(* PLC project Regular Expressions, CODESYS CODESYS V3.5 SP18 Patch 5 *)
(* stored: creationDateTime 2024-02-02T21:46:32.2565392, version 1.1.0.0, modificationDateTime 2024-02-02T18:21:46.8982597, organization GG *)
(* Regular Expressions - this is a simple implementation.

See the documentation folder for an introduction (the folder itself). *)

{attribute 'qualified_only'}
{attribute 'strict'}
TYPE eTokenType : (INVALID := 0, LITERAL, ANYCHAR, WILDCARD);
END_TYPE

TYPE typCompiledPattern : STRUCT
  xCaseInsensitive : BOOL;
  atTokens : ARRAY[0..ParameterList.uiMaxPatternTokens] OF typPatternToken;
  uiCountTokens : UINT;
END_STRUCT;
END_TYPE

TYPE typCompiledPatternW : STRUCT
  xCaseInsensitive : BOOL;
  atTokens : ARRAY[0..ParameterList.uiMaxPatternTokens] OF typPatternTokenW;
  uiCountTokens : UINT;
END_STRUCT;
END_TYPE

TYPE typPatternToken : STRUCT
  eType : eTokenType;
  bChar : BYTE;
  bAlternativeChar : BYTE;
END_STRUCT;
END_TYPE

TYPE typPatternTokenW : STRUCT
  eType : eTokenType;
  dwChar : DWORD;
  dwAlternativeChar : DWORD;
END_STRUCT;
END_TYPE

{attribute 'parameterlist'}
{attribute 'qualified_only'}
VAR_GLOBAL CONSTANT  (* ParameterList *)
  uiMaxPatternTokens : UINT := 255;  (* The maximum amount of tokens to support parsing (compiling) - the counting starts from 0, so add 1 to the number in your mind *)
END_VAR

(* Converts an ANSI/ISO 8859-1 compiled pattern to an Unicode compiled pattern. ANSI/ISO 8859-1 compiled patterns can be converted to Unicode without any loss. *)
FUNCTION FuCompiledPatternAnsiToW : typCompiledPatternW
  VAR_INPUT
    typPattern : typCompiledPattern;
  END_VAR
  VAR
    i : UDINT;
  END_VAR

            IF typPattern.uiCountTokens = 0 THEN
    RETURN;
END_IF

FuCompiledPatternAnsiToW.xCaseInsensitive := typPattern.xCaseInsensitive;
FuCompiledPatternAnsiToW.uiCountTokens := typPattern.uiCountTokens;

FOR i := 0 TO TO_UDINT((typPattern.uiCountTokens - 1)) BY 1 DO
    FuCompiledPatternAnsiToW.atTokens[i].eType := typPattern.atTokens[i].eType;
    FuCompiledPatternAnsiToW.atTokens[i].dwChar := TO_DWORD(typPattern.atTokens[i].bChar);
    FuCompiledPatternAnsiToW.atTokens[i].dwAlternativeChar := TO_DWORD(typPattern.atTokens[i].bAlternativeChar); 
END_FOR

          
END_FUNCTION

(* Compiles the pattern into a stream of tokens for matching. The ISO 8859-1 latin alphabet can be matched case insensitive, otherwise by default the pattern is case sensitive. A few examples of valid patterns: - 'A*bEd' - 'A*?bEd' - 'A.b*e*' - '*A\.b\*e*' - 'A?\bed' The return value signifies whether compilation was successful, or the given pattern is invalid. *)
{attribute 'qualified_only'}
FUNCTION FuCompilePattern : BOOL
  VAR_INPUT
    sPattern : STRING(255);  (* The pattern string to compile *)
    xCaseInsensitive : BOOL := FALSE;  (* Whether the pattern is case insensitive (ISO 8859-1 latin1) *)
  END_VAR
  VAR_OUTPUT
    typPattern : typCompiledPattern;  (* The compiled pattern, for "FuMatchExpression" *)
  END_VAR
  VAR
    i : UINT;
    tempChar : BYTE;
    tempNextChar : BYTE;
    tempIndex : UINT;
    tempMaxStrIndex : UINT;
  END_VAR
  VAR CONSTANT
    CHAR_WILDCARD : BYTE := 42;  (* * *)
    CHAR_LAZINESS : BYTE := 63;  (* ? *)
    CHAR_DOT : BYTE := 46;  (* . *)
    CHAR_ESCAPE : BYTE := 92;  (* \ *)
  END_VAR

            FuCompilePattern := FALSE;

IF sPattern = '' THEN
    RETURN;
END_IF

tempMaxStrIndex := TO_UINT(Standard.LEN(sPattern)) - 1;

FOR i := 0 TO tempMaxStrIndex BY 1 DO
    IF sPattern[i] = 0 OR_ELSE tempIndex > ParameterList.uiMaxPatternTokens THEN
        EXIT;
    END_IF
    
    tempChar := TO_BYTE(sPattern[i]);
    
    IF i < tempMaxStrIndex THEN
        tempNextChar := TO_BYTE(sPattern[(i + 1)]);
    ELSE
        tempNextChar := 0;
    END_IF
    
    IF tempChar = CHAR_WILDCARD THEN // Wildcard (*)
        typPattern.atTokens[tempIndex].eType := eTokenType.WILDCARD;
        typPattern.atTokens[tempIndex].bChar := 0; // Use bChar as modifier to be lazy
    ELSIF
        tempChar = CHAR_LAZINESS AND_THEN
        tempIndex > 0 AND_THEN
        typPattern.atTokens[(tempIndex - 1)].eType = eTokenType.WILDCARD
    THEN // Laziness (?), but only if previously wildcard, otherwise literal
        typPattern.atTokens[(tempIndex - 1)].bChar := 1;
        CONTINUE;
    ELSIF tempChar = CHAR_DOT THEN // Single char (.)
        typPattern.atTokens[tempIndex].eType := eTokenType.ANYCHAR;
    ELSIF
        tempChar = CHAR_ESCAPE AND_THEN (
            tempNextChar = CHAR_WILDCARD OR_ELSE
            tempNextChar = CHAR_DOT
        )
    THEN // Backslash (escape token for . or *, if followed by . or *)
        typPattern.atTokens[tempIndex].eType := eTokenType.LITERAL;
        typPattern.atTokens[tempIndex].bChar := tempNextChar;
        i := i + 1;
    ELSE
        typPattern.atTokens[tempIndex].eType := eTokenType.LITERAL;
        typPattern.atTokens[tempIndex].bChar := tempChar;
        
        tempNextChar := 0;
        IF xCaseInsensitive THEN
            // Calculate for the ISO 8859-1 latin1 alphabet the uppercase or lowercase character number
            IF tempChar >= 65 AND_THEN tempChar <= 90 THEN
                // Uppercase A-Z
                tempNextChar := tempChar + 32;
            ELSIF tempChar >= 97 AND_THEN tempChar <= 122 THEN
                // Lowercase a-z
                tempNextChar := tempChar - 32;
            ELSIF tempChar >= 192 AND_THEN tempChar <= 221 AND_THEN tempChar <> 215 THEN
                // Uppercase ISO 8859-1
                tempNextChar := tempChar + 32;
            ELSIF tempChar >= 224 AND_THEN tempChar <= 253 AND_THEN tempChar <> 247 THEN
                // Lowercase ISO 8859-1
                tempNextChar := tempChar - 32; 
            END_IF
        END_IF
        
        typPattern.atTokens[tempIndex].bAlternativeChar := tempNextChar;
    END_IF
    
    tempIndex := tempIndex + 1;
    typPattern.uiCountTokens := tempIndex;
END_FOR

FuCompilePattern := (tempIndex > 0);
typPattern.xCaseInsensitive := xCaseInsensitive;

          
END_FUNCTION

(* Compiles the pattern into a stream of tokens for matching. This is the UTF-8 version of FuCompilePattern. Disabling strict conformity allows the usage of the extended ASCII alphabet (ISO 8859-1, decimal 160-255), as long as it doesn't form a valid UTF-8 byte sequence. The alphabet can be matched case insensitive, otherwise by default the pattern is case sensitive. The case mapping table is NOT completely covered, as such you MAY encounter missing case conversion for some languages. A few examples of valid patterns: - 'A*bEd' - 'A*?bEd' - 'A.b*e*' - '*A\.b\*e*' - 'A?\bed' The return value signifies whether compilation was successful, or the given pattern is invalid. *)
{attribute 'qualified_only'}
FUNCTION FuCompilePatternUTF8 : BOOL
  VAR_INPUT
    psPattern : POINTER TO STRING(1);  (* The pattern string to compile - for technical reasons this is a STRING(1), although any length is supported *)
    udiPatternLength : UDINT;  (* Pattern string length (in bytes, not codepoints) *)
    xCaseInsensitive : BOOL := FALSE;  (* Whether the pattern is case insensitive *)
    xStrictConformity : BOOL := TRUE;  (* Require strict conformity to the Unicode standard *)
  END_VAR
  VAR_OUTPUT
    typPattern : typCompiledPatternW;  (* The compiled pattern, for "FuMatchExpressionUTF8" *)
  END_VAR
  VAR
    tempPointer : POINTER TO STRING(1);
    i : UDINT;
    tempChar : DWORD;
    tempCharLength : UDINT;
    tempNextChar : DWORD;
    tempNextCharLength : UDINT;
    tempIndex : UINT;
    tempMaxStrIndex : UDINT;
  END_VAR
  VAR CONSTANT
    CHAR_WILDCARD : DWORD := 42;  (* * *)
    CHAR_LAZINESS : DWORD := 63;  (* ? *)
    CHAR_DOT : DWORD := 46;  (* . *)
    CHAR_ESCAPE : DWORD := 92;  (* \ *)
  END_VAR

            FuCompilePatternUTF8 := FALSE;

IF udiPatternLength = 0 THEN
    RETURN;
END_IF

tempPointer := psPattern;

i := 0;
tempMaxStrIndex := udiPatternLength - 1;

WHILE i <= tempMaxStrIndex DO
    IF tempIndex > ParameterList.uiMaxPatternTokens THEN
        EXIT;
    END_IF
    
    IF
        NOT FuUtf8CharToDword(
            psInput := (tempPointer + i),
            udiStringLength := (udiPatternLength - i),
            xStrictConformity := xStrictConformity,
            dwCodepoint => tempChar,
            usiByteLength => tempCharLength
        )
    THEN
        RETURN;
    END_IF
    
    IF tempChar = 0 THEN
        EXIT;
    END_IF
    
    IF
        i > tempMaxStrIndex OR_ELSE
        NOT FuUtf8CharToDword(
            psInput := (tempPointer + i + tempCharLength),
            udiStringLength := (udiPatternLength - i),
            xStrictConformity := xStrictConformity,
            dwCodepoint => tempNextChar,
            usiByteLength => tempNextCharLength
        )
    THEN
        tempNextChar := 0;
        tempNextCharLength := 0;
    END_IF
    
    IF tempChar = CHAR_WILDCARD THEN // Wildcard (*)
        typPattern.atTokens[tempIndex].eType := eTokenType.WILDCARD;
        typPattern.atTokens[tempIndex].dwChar := 0; // Use dwChar as modifier to be lazy
    ELSIF
        tempChar = CHAR_LAZINESS AND_THEN
        tempIndex > 0 AND_THEN
        typPattern.atTokens[(tempIndex - 1)].eType = eTokenType.WILDCARD
    THEN // Laziness (?), but only if previously wildcard, otherwise literal
        typPattern.atTokens[(tempIndex - 1)].dwChar := 1;
        
        i := i + tempCharLength;
        CONTINUE;
    ELSIF tempChar = CHAR_DOT THEN // Single char (.)
        typPattern.atTokens[tempIndex].eType := eTokenType.ANYCHAR;
    ELSIF
        tempChar = CHAR_ESCAPE AND_THEN (
            tempNextChar = CHAR_WILDCARD OR_ELSE
            tempNextChar = CHAR_DOT
        )
    THEN // Backslash (escape token for . or *, if followed by . or *)
        typPattern.atTokens[tempIndex].eType := eTokenType.LITERAL;
        typPattern.atTokens[tempIndex].dwChar := tempNextChar;
        i := i + tempNextCharLength;
    ELSE
        typPattern.atTokens[tempIndex].eType := eTokenType.LITERAL;
        typPattern.atTokens[tempIndex].dwChar := tempChar;
        
        IF xCaseInsensitive THEN
            // Calculate for the ISO 8859-1 latin1 alphabet the uppercase or lowercase character number (efficient way)
            IF tempChar >= 65 AND_THEN tempChar <= 90 THEN
                // Uppercase A-Z
                tempNextChar := tempChar + 32;
            ELSIF tempChar >= 97 AND_THEN tempChar <= 122 THEN
                // Lowercase a-z
                tempNextChar := tempChar - 32;
            ELSIF tempChar >= 192 AND_THEN tempChar <= 221 AND_THEN tempChar <> 215 THEN
                // Uppercase ISO 8859-1
                tempNextChar := tempChar + 32;
            ELSIF tempChar >= 224 AND_THEN tempChar <= 253 AND_THEN tempChar <> 247 THEN
                // Lowercase ISO 8859-1
                tempNextChar := tempChar - 32; 
            ELSE
                // If we're not in the ISO 8859-1 latin1 alphabet range, use the Unicode function to calculate it
                tempNextChar := FuUnicodeCodepointCaseConvert(tempChar);
            END_IF
        ELSE
            tempNextChar := 0;
        END_IF
        
        typPattern.atTokens[tempIndex].dwAlternativeChar := tempNextChar;
    END_IF
    
    tempIndex := tempIndex + 1;
    typPattern.uiCountTokens := tempIndex;
    
    i := i + tempCharLength;
END_WHILE

FuCompilePatternUTF8 := (tempIndex > 0);
typPattern.xCaseInsensitive := xCaseInsensitive;

          
END_FUNCTION

(* Compiles the pattern into a stream of tokens for matching. This is the UTF-16 (WSTRING) version of FuCompilePattern. The alphabet can be matched case insensitive, otherwise by default the pattern is case sensitive. The case mapping table is NOT completely covered, as such you MAY encounter missing case conversion for some languages. A few examples of valid patterns: - 'A*bEd' - 'A*?bEd' - 'A.b*e*' - '*A\.b\*e*' - 'A?\bed' The return value signifies whether compilation was successful, or the given pattern is invalid. *)
{attribute 'qualified_only'}
FUNCTION FuCompilePatternW : BOOL
  VAR_INPUT
    pwsPattern : POINTER TO WSTRING(1);  (* The pattern string to compile - for technical reasons this is a WSTRING(1), although any length is supported *)
    udiPatternLength : UDINT;  (* Pattern string length (in words (length in bytes/2), not codepoints) *)
    xCaseInsensitive : BOOL := FALSE;  (* Whether the pattern is case insensitive *)
  END_VAR
  VAR_OUTPUT
    typPattern : typCompiledPatternW;  (* The compiled pattern, for "FuMatchExpressionW" *)
  END_VAR
  VAR
    tempPointer : POINTER TO WSTRING(1);
    i : UDINT;
    tempChar : DWORD;
    tempCharLength : UDINT;
    tempNextChar : DWORD;
    tempNextCharLength : UDINT;
    tempIndex : UINT;
    tempMaxStrIndex : UDINT;
  END_VAR
  VAR CONSTANT
    CHAR_WILDCARD : DWORD := 42;  (* * *)
    CHAR_LAZINESS : DWORD := 63;  (* ? *)
    CHAR_DOT : DWORD := 46;  (* . *)
    CHAR_ESCAPE : DWORD := 92;  (* \ *)
  END_VAR

            FuCompilePatternW := FALSE;

IF udiPatternLength = 0 THEN
    RETURN;
END_IF

tempPointer := pwsPattern;

i := 0;
tempMaxStrIndex := udiPatternLength - 1;

WHILE i <= tempMaxStrIndex DO
    IF tempIndex > ParameterList.uiMaxPatternTokens THEN
        EXIT;
    END_IF
    
    IF NOT FuUtf16CharToDword(psInput := (tempPointer + (i * 2)), udiStringLength := (udiPatternLength - (i * 2)), dwCodepoint => tempChar, usiWordLength => tempCharLength) THEN
        RETURN;
    END_IF
    
    IF tempChar = 0 THEN
        EXIT;
    END_IF
    
    IF
        i > tempMaxStrIndex OR_ELSE
        NOT FuUtf16CharToDword(
            psInput := (tempPointer + (i * 2) + (tempCharLength * 2)),
            udiStringLength := (udiPatternLength - (i * 2) - (tempCharLength * 2)),
            dwCodepoint => tempNextChar,
            usiWordLength => tempNextCharLength
        )
    THEN
        tempNextChar := 0;
        tempNextCharLength := 0;
    END_IF
    
    IF tempChar = CHAR_WILDCARD THEN // Wildcard (*)
        typPattern.atTokens[tempIndex].eType := eTokenType.WILDCARD;
        typPattern.atTokens[tempIndex].dwChar := 0; // Use dwChar as modifier to be lazy
    ELSIF
        tempChar = CHAR_LAZINESS AND_THEN
        tempIndex > 0 AND_THEN
        typPattern.atTokens[(tempIndex - 1)].eType = eTokenType.WILDCARD
    THEN // Laziness (?), but only if previously wildcard, otherwise literal
        typPattern.atTokens[(tempIndex - 1)].dwChar := 1;
        
        i := i + tempCharLength;
        CONTINUE;
    ELSIF tempChar = CHAR_DOT THEN // Single char (.)
        typPattern.atTokens[tempIndex].eType := eTokenType.ANYCHAR;
    ELSIF
        tempChar = CHAR_ESCAPE AND_THEN (
            tempNextChar = CHAR_WILDCARD OR_ELSE
            tempNextChar = CHAR_DOT
        )
    THEN // Backslash (escape token for . or *, if followed by . or *)
        typPattern.atTokens[tempIndex].eType := eTokenType.LITERAL;
        typPattern.atTokens[tempIndex].dwChar := tempNextChar;
        i := i + tempNextCharLength;
    ELSE
        typPattern.atTokens[tempIndex].eType := eTokenType.LITERAL;
        typPattern.atTokens[tempIndex].dwChar := tempChar;
        
        IF xCaseInsensitive THEN
            // Calculate for the ISO 8859-1 latin1 alphabet the uppercase or lowercase character number (efficient way)
            IF tempChar >= 65 AND_THEN tempChar <= 90 THEN
                // Uppercase A-Z
                tempNextChar := tempChar + 32;
            ELSIF tempChar >= 97 AND_THEN tempChar <= 122 THEN
                // Lowercase a-z
                tempNextChar := tempChar - 32;
            ELSIF tempChar >= 192 AND_THEN tempChar <= 221 AND_THEN tempChar <> 215 THEN
                // Uppercase ISO 8859-1
                tempNextChar := tempChar + 32;
            ELSIF tempChar >= 224 AND_THEN tempChar <= 253 AND_THEN tempChar <> 247 THEN
                // Lowercase ISO 8859-1
                tempNextChar := tempChar - 32; 
            ELSE
                // If we're not in the ISO 8859-1 latin1 alphabet range, use the UTF-8 function to calculate it
                tempNextChar := FuUnicodeCodepointCaseConvert(tempChar);
            END_IF
        ELSE
            tempNextChar := 0;
        END_IF
        
        typPattern.atTokens[tempIndex].dwAlternativeChar := tempNextChar;
    END_IF
    
    tempIndex := tempIndex + 1;
    typPattern.uiCountTokens := tempIndex;
    
    i := i + tempCharLength;
END_WHILE

FuCompilePatternW := (tempIndex > 0);
typPattern.xCaseInsensitive := xCaseInsensitive;

          
END_FUNCTION

(* Same as FuCompilePatternW, except it doesn't take a pointer and has a fixed length. *)
{attribute 'qualified_only'}
FUNCTION FuCompilePatternW2 : BOOL
  VAR_INPUT
    wsPattern : WSTRING(255);  (* The pattern string to compile *)
    xCaseInsensitive : BOOL := FALSE;  (* Whether the pattern is case insensitive *)
  END_VAR
  VAR_OUTPUT
    typPattern : typCompiledPatternW;  (* The compiled pattern, for "FuMatchExpressionW" *)
  END_VAR

            FuCompilePatternW2 := FuCompilePatternW(ADR(wsPattern), TO_UDINT(Stu.StrLenW(ADR(wsPattern))), xCaseInsensitive, typPattern => typPattern);

          
END_FUNCTION

(* Matches the given compiled pattern against the subject. *)
{attribute 'qualified_only'}
FUNCTION FuMatchExpression : BOOL
  VAR_INPUT
    typPattern : typCompiledPattern;  (* The compiled pattern from "FuCompilePattern" *)
    psSubject : POINTER TO STRING(1);  (* A pointer to the subject string - for technical reasons this is a STRING(1), although any size is supported *)
    udiLength : UDINT;  (* The length of the subject string *)
  END_VAR
  VAR
    tempPtrStr : POINTER TO BYTE;
    tempPtrStrMatching : POINTER TO BYTE;
    tempStrIndex : UDINT;
    tempStrIndexMatching : UDINT;
    i : UINT;
    j : UINT;
    k : LINT;
    tempLaziness : BOOL;
    tempHasEndChar : BOOL;
    tempEndChar : BYTE;
    tempEndChar2 : BYTE;
    tempWildcardSearchStart : LINT;
    tempWildcardSearchEnd : LINT;
    tempWildcardSearchBy : LINT;
    tempWildcardSearchSuccess : BOOL;
  END_VAR

            FuMatchExpression := FALSE;

IF typPattern.uiCountTokens = 0 OR_ELSE udiLength = 0 THEN
    RETURN;
END_IF

tempPtrStr := psSubject;
tempStrIndex := 0;

WHILE i < typPattern.uiCountTokens DO
    IF tempStrIndex >= udiLength THEN
        // Only if all following tokens are of type WILDCARD, we can allow a match to be positive
        FOR j := i TO (typPattern.uiCountTokens - 1) BY 1 DO
            IF typPattern.atTokens[j].eType <> eTokenType.WILDCARD THEN
                FuMatchExpression := FALSE;
                RETURN;
            END_IF
        END_FOR
        
        FuMatchExpression := TRUE;
        RETURN;
    END_IF
    
    CASE typPattern.atTokens[i].eType OF
        eTokenType.INVALID: // We shouldn't ever get an invalid token inside our token array that isn't behind our count
            RETURN;
        
        eTokenType.LITERAL:
            IF
                tempPtrStr[tempStrIndex] <> typPattern.atTokens[i].bChar AND_THEN
                (
                    NOT typPattern.xCaseInsensitive OR_ELSE (
                        typPattern.atTokens[i].bAlternativeChar <> 0 AND_THEN
                        tempPtrStr[tempStrIndex] <> typPattern.atTokens[i].bAlternativeChar
                    )
                )
            THEN
                RETURN;
            END_IF
            
            tempStrIndex := tempStrIndex + 1;
        
        eTokenType.ANYCHAR:
            tempStrIndex := tempStrIndex + 1;
        
        eTokenType.WILDCARD:
            tempLaziness := (typPattern.atTokens[i].bChar = 1);
            tempHasEndChar := FALSE;
            
            FOR j := i + 1 TO (typPattern.uiCountTokens - 1) BY 1 DO
                IF typPattern.atTokens[j].eType = eTokenType.LITERAL THEN
                    tempHasEndChar := TRUE;
                    tempEndChar := typPattern.atTokens[j].bChar;
                    tempEndChar2 := typPattern.atTokens[j].bAlternativeChar;
                    EXIT;
                END_IF
            END_FOR
            
            // If we don't have any characters to match on at the end of the pattern, we match immediately
            IF NOT tempHasEndChar THEN
                FuMatchExpression := TRUE;
                RETURN;
            END_IF
            
            IF tempLaziness THEN
                // Advance token pointer once more because the next token is the laziness token we already used
                i := i + 1;
                
                // If the wildcard is lazy, search from front to back
                tempWildcardSearchStart := TO_LINT(tempStrIndex);
                tempWildcardSearchEnd := TO_LINT(udiLength);
                tempWildcardSearchBy := 1;
            ELSE
                // If the wildcard is NOT lazy, search from back to front (greedy!)
                tempWildcardSearchStart := TO_LINT(udiLength);
                tempWildcardSearchEnd := TO_LINT(tempStrIndex);
                tempWildcardSearchBy := -1;
            END_IF
            
            tempWildcardSearchSuccess := FALSE;
            FOR k := tempWildcardSearchStart TO tempWildcardSearchEnd BY tempWildcardSearchBy DO
                IF
                    tempPtrStr[k] = tempEndChar OR_ELSE
                    (typPattern.xCaseInsensitive AND_THEN tempEndChar2 <> 0 AND_THEN tempPtrStr[k] = tempEndChar2)
                THEN
                    tempWildcardSearchSuccess := TRUE;
                    tempStrIndex := TO_UDINT(k);
                    EXIT;
                END_IF
            END_FOR
            
            IF NOT tempWildcardSearchSuccess THEN
                RETURN;
            END_IF
    END_CASE
    
    i := i + 1;
END_WHILE

FuMatchExpression := (tempStrIndex >= udiLength);

          
END_FUNCTION

(* Matches the given compiled pattern against the subject. This is the UTF-8 version of FuMatchExpression. Disabling strict conformity allows the usage of the extended ASCII alphabet (ISO 8859-1, decimal 160-255), as long as it doesn't form a valid UTF-8 byte sequence. *)
{attribute 'qualified_only'}
FUNCTION FuMatchExpressionUTF8 : BOOL
  VAR_INPUT
    typPattern : typCompiledPatternW;  (* The compiled pattern from "FuCompilePatternW" *)
    psSubject : POINTER TO STRING(1);  (* A pointer to the subject string - for technical reasons this is a STRING(1), although any size is supported *)
    udiLength : UDINT;  (* The length of the subject string (in bytes, not codepoints) *)
    xStrictConformity : BOOL := TRUE;  (* Require strict conformity to the Unicode standard *)
  END_VAR
  VAR
    tempPtrStr : POINTER TO BYTE;
    tempPtrStrMatching : POINTER TO BYTE;
    tempStrIndex : UDINT;
    tempStrIndexMatching : UDINT;
    i : UINT;
    j : UINT;
    k : LINT;
    tempChar : DWORD;
    tempCharLength : USINT;
    tempNextChar : DWORD;
    tempNextCharLength : DWORD;
    tempLaziness : BOOL;
    tempHasEndChar : BOOL;
    tempEndChar : DWORD;
    tempEndChar2 : DWORD;
    tempWildcardSearchStart : LINT;
    tempWildcardSearchEnd : LINT;
    tempWildcardSearchBy : LINT;
    tempWildcardSearchOffset : UDINT;
    tempWildcardSearchSuccess : BOOL;
  END_VAR

            FuMatchExpressionUTF8 := FALSE;

IF typPattern.uiCountTokens = 0 OR_ELSE udiLength = 0 THEN
    RETURN;
END_IF

tempPtrStr := psSubject;
tempStrIndex := 0;

WHILE i < typPattern.uiCountTokens DO
    IF tempStrIndex >= udiLength THEN
        // Only if all following tokens are of type WILDCARD, we can allow a match to be positive
        FOR j := i TO (typPattern.uiCountTokens - 1) BY 1 DO
            IF typPattern.atTokens[j].eType <> eTokenType.WILDCARD THEN
                FuMatchExpressionUTF8 := FALSE;
                RETURN;
            END_IF
        END_FOR
        
        FuMatchExpressionUTF8 := TRUE;
        RETURN;
    END_IF
    
    IF
        NOT FuUtf8CharToDword(
            psInput := (tempPtrStr + tempStrIndex),
            udiStringLength := (udiLength - tempStrIndex),
            xStrictConformity := xStrictConformity,
            dwCodepoint => tempChar,
            usiByteLength => tempCharLength
        )
    THEN
        RETURN;
    END_IF
    
    CASE typPattern.atTokens[i].eType OF
        eTokenType.INVALID: // We shouldn't ever get an invalid token inside our token array that isn't behind our count
            RETURN;
        
        eTokenType.LITERAL:
            IF
                tempChar <> typPattern.atTokens[i].dwChar AND_THEN
                (
                    NOT typPattern.xCaseInsensitive OR_ELSE
                    typPattern.atTokens[i].dwAlternativeChar = 0 OR_ELSE
                    tempChar <> typPattern.atTokens[i].dwAlternativeChar
                ) 
            THEN
                RETURN;
            END_IF
            
            tempStrIndex := tempStrIndex + tempCharLength;
        
        eTokenType.ANYCHAR:
            tempStrIndex := tempStrIndex + tempCharLength;
        
        eTokenType.WILDCARD:
            tempLaziness := (typPattern.atTokens[i].dwChar = 1);
            tempHasEndChar := FALSE;
            
            FOR j := i + 1 TO (typPattern.uiCountTokens - 1) BY 1 DO
                IF typPattern.atTokens[j].eType = eTokenType.LITERAL THEN
                    tempHasEndChar := TRUE;
                    tempEndChar := typPattern.atTokens[j].dwChar;
                    tempEndChar2 := typPattern.atTokens[j].dwAlternativeChar;
                    EXIT;
                END_IF
            END_FOR
            
            // If we don't have any characters to match on at the end of the pattern, we match immediately
            IF NOT tempHasEndChar THEN
                FuMatchExpressionUTF8 := TRUE;
                RETURN;
            END_IF
            
            IF tempLaziness THEN
                // Advance token pointer once more because the next token is the laziness token we already used
                i := i + 1;
                
                // If the wildcard is lazy, search from front to back
                tempWildcardSearchStart := TO_LINT(tempStrIndex);
                tempWildcardSearchEnd := TO_LINT(udiLength);
                tempWildcardSearchBy := 1;
            ELSE
                // If the wildcard is NOT lazy, search from back to front (greedy!)
                tempWildcardSearchStart := TO_LINT(udiLength);
                tempWildcardSearchEnd := TO_LINT(tempStrIndex);
                tempWildcardSearchBy := -1;
            END_IF
            
            tempWildcardSearchSuccess := FALSE;
            tempWildcardSearchOffset := 0;
            
            FOR k := tempWildcardSearchStart TO tempWildcardSearchEnd BY tempWildcardSearchBy DO
                IF
                    FuUtf8CharToDword(
                        psInput := (tempPtrStr + LINT_TO___XWORD(k)),
                        udiStringLength := (udiLength - tempWildcardSearchOffset),
                        xStrictConformity := xStrictConformity,
                        dwCodepoint => tempNextChar,
                        usiByteLength => tempNextCharLength
                    )
                THEN
                    tempWildcardSearchOffset := tempWildcardSearchOffset + tempNextCharLength;
                    
                    IF
                        tempNextChar = tempEndChar OR_ELSE
                        (typPattern.xCaseInsensitive AND_THEN tempEndChar2 <> 0 AND_THEN tempNextChar = tempEndChar2)
                    THEN
                        tempWildcardSearchSuccess := TRUE;
                        tempStrIndex := TO_UDINT(k);
                        EXIT;
                    END_IF
                ELSE
                    tempWildcardSearchOffset := tempWildcardSearchOffset + 1;
                END_IF
            END_FOR
            
            IF NOT tempWildcardSearchSuccess THEN
                RETURN;
            END_IF
    END_CASE
    
    i := i + 1;
END_WHILE

FuMatchExpressionUTF8 := (tempStrIndex >= udiLength);

          
END_FUNCTION

(* Matches the given compiled pattern against the subject. This is the UTF-16 (WSTRING) version of FuMatchExpression. *)
{attribute 'qualified_only'}
FUNCTION FuMatchExpressionW : BOOL
  VAR_INPUT
    typPattern : typCompiledPatternW;  (* The compiled pattern from "FuCompilePatternW" *)
    pwsSubject : POINTER TO WSTRING(1);  (* A pointer to the subject string - for technical reasons this is a WSTRING(1), although any size is supported *)
    udiLength : UDINT;  (* The length of the subject string (in words (length in bytes/2), not codepoints) *)
  END_VAR
  VAR
    tempPtrStr : POINTER TO WORD;
    tempPtrStrMatching : POINTER TO WORD;
    tempStrIndex : UDINT;
    tempStrIndexMatching : UDINT;
    i : UINT;
    j : UINT;
    k : LINT;
    tempChar : DWORD;
    tempCharLength : USINT;
    tempNextChar : DWORD;
    tempNextCharLength : DWORD;
    tempLaziness : BOOL;
    tempHasEndChar : BOOL;
    tempEndChar : DWORD;
    tempEndChar2 : DWORD;
    tempWildcardSearchStart : LINT;
    tempWildcardSearchEnd : LINT;
    tempWildcardSearchBy : LINT;
    tempWildcardSearchOffset : UDINT;
    tempWildcardSearchSuccess : BOOL;
  END_VAR

            FuMatchExpressionW := FALSE;

IF typPattern.uiCountTokens = 0 OR_ELSE udiLength = 0 THEN
    RETURN;
END_IF

tempPtrStr := pwsSubject;
tempStrIndex := 0;

WHILE i < typPattern.uiCountTokens DO
    IF tempStrIndex >= udiLength THEN
        // Only if all following tokens are of type WILDCARD, we can allow a match to be positive
        FOR j := i TO (typPattern.uiCountTokens - 1) BY 1 DO
            IF typPattern.atTokens[j].eType <> eTokenType.WILDCARD THEN
                FuMatchExpressionW := FALSE;
                RETURN;
            END_IF
        END_FOR
        
        FuMatchExpressionW := TRUE;
        RETURN;
    END_IF
    
    IF NOT FuUtf16CharToDword(psInput := (tempPtrStr + (tempStrIndex * 2)), udiStringLength := (udiLength - (tempStrIndex * 2)), dwCodepoint => tempChar, usiWordLength => tempCharLength) THEN
        RETURN;
    END_IF
    
    CASE typPattern.atTokens[i].eType OF
        eTokenType.INVALID: // We shouldn't ever get an invalid token inside our token array that isn't behind our count
            RETURN;
        
        eTokenType.LITERAL:
            IF
                tempChar <> typPattern.atTokens[i].dwChar AND_THEN
                (
                    NOT typPattern.xCaseInsensitive OR_ELSE
                    typPattern.atTokens[i].dwAlternativeChar = 0 OR_ELSE
                    tempChar <> typPattern.atTokens[i].dwAlternativeChar
                ) 
            THEN
                RETURN;
            END_IF
            
            tempStrIndex := tempStrIndex + tempCharLength;
        
        eTokenType.ANYCHAR:
            tempStrIndex := tempStrIndex + tempCharLength;
        
        eTokenType.WILDCARD:
            tempLaziness := (typPattern.atTokens[i].dwChar = 1);
            tempHasEndChar := FALSE;
            
            FOR j := i + 1 TO (typPattern.uiCountTokens - 1) BY 1 DO
                IF typPattern.atTokens[j].eType = eTokenType.LITERAL THEN
                    tempHasEndChar := TRUE;
                    tempEndChar := typPattern.atTokens[j].dwChar;
                    tempEndChar2 := typPattern.atTokens[j].dwAlternativeChar;
                    EXIT;
                END_IF
            END_FOR
            
            // If we don't have any characters to match on at the end of the pattern, we match immediately
            IF NOT tempHasEndChar THEN
                FuMatchExpressionW := TRUE;
                RETURN;
            END_IF
            
            IF tempLaziness THEN
                // Advance token pointer once more because the next token is the laziness token we already used
                i := i + 1;
                
                // If the wildcard is lazy, search from front to back
                tempWildcardSearchStart := TO_LINT(tempStrIndex);
                tempWildcardSearchEnd := TO_LINT(udiLength);
                tempWildcardSearchBy := 1;
            ELSE
                // If the wildcard is NOT lazy, search from back to front (greedy!)
                tempWildcardSearchStart := TO_LINT(udiLength);
                tempWildcardSearchEnd := TO_LINT(tempStrIndex);
                tempWildcardSearchBy := -1;
            END_IF
            
            tempWildcardSearchSuccess := FALSE;
            tempWildcardSearchOffset := 0;
            
            FOR k := tempWildcardSearchStart TO tempWildcardSearchEnd BY tempWildcardSearchBy DO
                IF
                    FuUtf16CharToDword(
                        psInput := (tempPtrStr + LINT_TO___XWORD(k)),
                        udiStringLength := (udiLength - tempWildcardSearchOffset),
                        dwCodepoint => tempNextChar,
                        usiWordLength => tempNextCharLength
                    )
                THEN
                    tempWildcardSearchOffset := tempWildcardSearchOffset + tempNextCharLength;
                    
                    IF
                        tempNextChar = tempEndChar OR_ELSE
                        (typPattern.xCaseInsensitive AND_THEN tempEndChar2 <> 0 AND_THEN tempNextChar = tempEndChar2)
                    THEN
                        tempWildcardSearchSuccess := TRUE;
                        tempStrIndex := TO_UDINT(k);
                        EXIT;
                    END_IF
                ELSE
                    tempWildcardSearchOffset := tempWildcardSearchOffset + 1;
                END_IF
            END_FOR
            
            IF NOT tempWildcardSearchSuccess THEN
                RETURN;
            END_IF
    END_CASE
    
    i := i + 1;
END_WHILE

FuMatchExpressionW := (tempStrIndex >= udiLength);

          
END_FUNCTION

(* Converts the given Unicode odepoint to the lowercase or uppercase codepoint (the opposite casing). If there is no codepoint mapping, then it will return 0. *)
{attribute 'qualified_only'}
FUNCTION FuUnicodeCodepointCaseConvert : DWORD
  VAR_INPUT
    dwCodepoint : DWORD;
  END_VAR

            FuUnicodeCodepointCaseConvert := 0;

// The following code has been generated from Unicode's UnicodeData.txt file
CASE dwCodepoint OF
    65:
        FuUnicodeCodepointCaseConvert := 97;
        RETURN;
    66:
        FuUnicodeCodepointCaseConvert := 98;
        RETURN;
    67:
        FuUnicodeCodepointCaseConvert := 99;
        RETURN;
    68:
        FuUnicodeCodepointCaseConvert := 100;
        RETURN;
    69:
        FuUnicodeCodepointCaseConvert := 101;
        RETURN;
    70:
        FuUnicodeCodepointCaseConvert := 102;
        RETURN;
    71:
        FuUnicodeCodepointCaseConvert := 103;
        RETURN;
    72:
        FuUnicodeCodepointCaseConvert := 104;
        RETURN;
    73:
        FuUnicodeCodepointCaseConvert := 105;
        RETURN;
    74:
        FuUnicodeCodepointCaseConvert := 106;
        RETURN;
    75:
        FuUnicodeCodepointCaseConvert := 107;
        RETURN;
    76:
        FuUnicodeCodepointCaseConvert := 108;
        RETURN;
    77:
        FuUnicodeCodepointCaseConvert := 109;
        RETURN;
    78:
        FuUnicodeCodepointCaseConvert := 110;
        RETURN;
    79:
        FuUnicodeCodepointCaseConvert := 111;
        RETURN;
    80:
        FuUnicodeCodepointCaseConvert := 112;
        RETURN;
    81:
        FuUnicodeCodepointCaseConvert := 113;
        RETURN;
    82:
        FuUnicodeCodepointCaseConvert := 114;
        RETURN;
    83:
        FuUnicodeCodepointCaseConvert := 115;
        RETURN;
    84:
        FuUnicodeCodepointCaseConvert := 116;
        RETURN;
    85:
        FuUnicodeCodepointCaseConvert := 117;
        RETURN;
    86:
        FuUnicodeCodepointCaseConvert := 118;
        RETURN;
    87:
        FuUnicodeCodepointCaseConvert := 119;
        RETURN;
    88:
        FuUnicodeCodepointCaseConvert := 120;
        RETURN;
    89:
        FuUnicodeCodepointCaseConvert := 121;
        RETURN;
    90:
        FuUnicodeCodepointCaseConvert := 122;
        RETURN;
    97:
        FuUnicodeCodepointCaseConvert := 65;
        RETURN;
    98:
        FuUnicodeCodepointCaseConvert := 66;
        RETURN;
    99:
        FuUnicodeCodepointCaseConvert := 67;
        RETURN;
    100:
        FuUnicodeCodepointCaseConvert := 68;
        RETURN;
    101:
        FuUnicodeCodepointCaseConvert := 69;
        RETURN;
    102:
        FuUnicodeCodepointCaseConvert := 70;
        RETURN;
    103:
        FuUnicodeCodepointCaseConvert := 71;
        RETURN;
    104:
        FuUnicodeCodepointCaseConvert := 72;
        RETURN;
    105:
        FuUnicodeCodepointCaseConvert := 73;
        RETURN;
    106:
        FuUnicodeCodepointCaseConvert := 74;
        RETURN;
    107:
        FuUnicodeCodepointCaseConvert := 75;
        RETURN;
    108:
        FuUnicodeCodepointCaseConvert := 76;
        RETURN;
    109:
        FuUnicodeCodepointCaseConvert := 77;
        RETURN;
    110:
        FuUnicodeCodepointCaseConvert := 78;
        RETURN;
    111:
        FuUnicodeCodepointCaseConvert := 79;
        RETURN;
    112:
        FuUnicodeCodepointCaseConvert := 80;
        RETURN;
    113:
        FuUnicodeCodepointCaseConvert := 81;
        RETURN;
    114:
        FuUnicodeCodepointCaseConvert := 82;
        RETURN;
    115:
        FuUnicodeCodepointCaseConvert := 83;
        RETURN;
    116:
        FuUnicodeCodepointCaseConvert := 84;
        RETURN;
    117:
        FuUnicodeCodepointCaseConvert := 85;
        RETURN;
    118:
        FuUnicodeCodepointCaseConvert := 86;
        RETURN;
    119:
        FuUnicodeCodepointCaseConvert := 87;
        RETURN;
    120:
        FuUnicodeCodepointCaseConvert := 88;
        RETURN;
    121:
        FuUnicodeCodepointCaseConvert := 89;
        RETURN;
    122:
        FuUnicodeCodepointCaseConvert := 90;
        RETURN;
    181:
        FuUnicodeCodepointCaseConvert := 924;
        RETURN;
    192:
        FuUnicodeCodepointCaseConvert := 224;
        RETURN;
    193:
        FuUnicodeCodepointCaseConvert := 225;
        RETURN;
    194:
        FuUnicodeCodepointCaseConvert := 226;
        RETURN;
    195:
        FuUnicodeCodepointCaseConvert := 227;
        RETURN;
    196:
        FuUnicodeCodepointCaseConvert := 228;
        RETURN;
    197:
        FuUnicodeCodepointCaseConvert := 229;
        RETURN;
    198:
        FuUnicodeCodepointCaseConvert := 230;
        RETURN;
    199:
        FuUnicodeCodepointCaseConvert := 231;
        RETURN;
    200:
        FuUnicodeCodepointCaseConvert := 232;
        RETURN;
    201:
        FuUnicodeCodepointCaseConvert := 233;
        RETURN;
    202:
        FuUnicodeCodepointCaseConvert := 234;
        RETURN;
    203:
        FuUnicodeCodepointCaseConvert := 235;
        RETURN;
    204:
        FuUnicodeCodepointCaseConvert := 236;
        RETURN;
    205:
        FuUnicodeCodepointCaseConvert := 237;
        RETURN;
    206:
        FuUnicodeCodepointCaseConvert := 238;
        RETURN;
    207:
        FuUnicodeCodepointCaseConvert := 239;
        RETURN;
    208:
        FuUnicodeCodepointCaseConvert := 240;
        RETURN;
    209:
        FuUnicodeCodepointCaseConvert := 241;
        RETURN;
    210:
        FuUnicodeCodepointCaseConvert := 242;
        RETURN;
    211:
        FuUnicodeCodepointCaseConvert := 243;
        RETURN;
    212:
        FuUnicodeCodepointCaseConvert := 244;
        RETURN;
    213:
        FuUnicodeCodepointCaseConvert := 245;
        RETURN;
    214:
        FuUnicodeCodepointCaseConvert := 246;
        RETURN;
    216:
        FuUnicodeCodepointCaseConvert := 248;
        RETURN;
    217:
        FuUnicodeCodepointCaseConvert := 249;
        RETURN;
    218:
        FuUnicodeCodepointCaseConvert := 250;
        RETURN;
    219:
        FuUnicodeCodepointCaseConvert := 251;
        RETURN;
    220:
        FuUnicodeCodepointCaseConvert := 252;
        RETURN;
    221:
        FuUnicodeCodepointCaseConvert := 253;
        RETURN;
    222:
        FuUnicodeCodepointCaseConvert := 254;
        RETURN;
    224:
        FuUnicodeCodepointCaseConvert := 192;
        RETURN;
    225:
        FuUnicodeCodepointCaseConvert := 193;
        RETURN;
    226:
        FuUnicodeCodepointCaseConvert := 194;
        RETURN;
    227:
        FuUnicodeCodepointCaseConvert := 195;
        RETURN;
    228:
        FuUnicodeCodepointCaseConvert := 196;
        RETURN;
    229:
        FuUnicodeCodepointCaseConvert := 197;
        RETURN;
    230:
        FuUnicodeCodepointCaseConvert := 198;
        RETURN;
    231:
        FuUnicodeCodepointCaseConvert := 199;
        RETURN;
    232:
        FuUnicodeCodepointCaseConvert := 200;
        RETURN;
    233:
        FuUnicodeCodepointCaseConvert := 201;
        RETURN;
    234:
        FuUnicodeCodepointCaseConvert := 202;
        RETURN;
    235:
        FuUnicodeCodepointCaseConvert := 203;
        RETURN;
    236:
        FuUnicodeCodepointCaseConvert := 204;
        RETURN;
    237:
        FuUnicodeCodepointCaseConvert := 205;
        RETURN;
    238:
        FuUnicodeCodepointCaseConvert := 206;
        RETURN;
    239:
        FuUnicodeCodepointCaseConvert := 207;
        RETURN;
    240:
        FuUnicodeCodepointCaseConvert := 208;
        RETURN;
    241:
        FuUnicodeCodepointCaseConvert := 209;
        RETURN;
    242:
        FuUnicodeCodepointCaseConvert := 210;
        RETURN;
    243:
        FuUnicodeCodepointCaseConvert := 211;
        RETURN;
    244:
        FuUnicodeCodepointCaseConvert := 212;
        RETURN;
    245:
        FuUnicodeCodepointCaseConvert := 213;
        RETURN;
    246:
        FuUnicodeCodepointCaseConvert := 214;
        RETURN;
    248:
        FuUnicodeCodepointCaseConvert := 216;
        RETURN;
    249:
        FuUnicodeCodepointCaseConvert := 217;
        RETURN;
    250:
        FuUnicodeCodepointCaseConvert := 218;
        RETURN;
    251:
        FuUnicodeCodepointCaseConvert := 219;
        RETURN;
    252:
        FuUnicodeCodepointCaseConvert := 220;
        RETURN;
    253:
        FuUnicodeCodepointCaseConvert := 221;
        RETURN;
    254:
        FuUnicodeCodepointCaseConvert := 222;
        RETURN;
    255:
        FuUnicodeCodepointCaseConvert := 376;
        RETURN;
    256:
        FuUnicodeCodepointCaseConvert := 257;
        RETURN;
    257:
        FuUnicodeCodepointCaseConvert := 256;
        RETURN;
    258:
        FuUnicodeCodepointCaseConvert := 259;
        RETURN;
    259:
        FuUnicodeCodepointCaseConvert := 258;
        RETURN;
    260:
        FuUnicodeCodepointCaseConvert := 261;
        RETURN;
    261:
        FuUnicodeCodepointCaseConvert := 260;
        RETURN;
    262:
        FuUnicodeCodepointCaseConvert := 263;
        RETURN;
    263:
        FuUnicodeCodepointCaseConvert := 262;
        RETURN;
    264:
        FuUnicodeCodepointCaseConvert := 265;
        RETURN;
    265:
        FuUnicodeCodepointCaseConvert := 264;
        RETURN;
    266:
        FuUnicodeCodepointCaseConvert := 267;
        RETURN;
    267:
        FuUnicodeCodepointCaseConvert := 266;
        RETURN;
    268:
        FuUnicodeCodepointCaseConvert := 269;
        RETURN;
    269:
        FuUnicodeCodepointCaseConvert := 268;
        RETURN;
    270:
        FuUnicodeCodepointCaseConvert := 271;
        RETURN;
    271:
        FuUnicodeCodepointCaseConvert := 270;
        RETURN;
    272:
        FuUnicodeCodepointCaseConvert := 273;
        RETURN;
    273:
        FuUnicodeCodepointCaseConvert := 272;
        RETURN;
    274:
        FuUnicodeCodepointCaseConvert := 275;
        RETURN;
    275:
        FuUnicodeCodepointCaseConvert := 274;
        RETURN;
    276:
        FuUnicodeCodepointCaseConvert := 277;
        RETURN;
    277:
        FuUnicodeCodepointCaseConvert := 276;
        RETURN;
    278:
        FuUnicodeCodepointCaseConvert := 279;
        RETURN;
    279:
        FuUnicodeCodepointCaseConvert := 278;
        RETURN;
    280:
        FuUnicodeCodepointCaseConvert := 281;
        RETURN;
    281:
        FuUnicodeCodepointCaseConvert := 280;
        RETURN;
    282:
        FuUnicodeCodepointCaseConvert := 283;
        RETURN;
    283:
        FuUnicodeCodepointCaseConvert := 282;
        RETURN;
    284:
        FuUnicodeCodepointCaseConvert := 285;
        RETURN;
    285:
        FuUnicodeCodepointCaseConvert := 284;
        RETURN;
    286:
        FuUnicodeCodepointCaseConvert := 287;
        RETURN;
    287:
        FuUnicodeCodepointCaseConvert := 286;
        RETURN;
    288:
        FuUnicodeCodepointCaseConvert := 289;
        RETURN;
    289:
        FuUnicodeCodepointCaseConvert := 288;
        RETURN;
    290:
        FuUnicodeCodepointCaseConvert := 291;
        RETURN;
    291:
        FuUnicodeCodepointCaseConvert := 290;
        RETURN;
    292:
        FuUnicodeCodepointCaseConvert := 293;
        RETURN;
    293:
        FuUnicodeCodepointCaseConvert := 292;
        RETURN;
    294:
        FuUnicodeCodepointCaseConvert := 295;
        RETURN;
    295:
        FuUnicodeCodepointCaseConvert := 294;
        RETURN;
    296:
        FuUnicodeCodepointCaseConvert := 297;
        RETURN;
    297:
        FuUnicodeCodepointCaseConvert := 296;
        RETURN;
    298:
        FuUnicodeCodepointCaseConvert := 299;
        RETURN;
    299:
        FuUnicodeCodepointCaseConvert := 298;
        RETURN;
    300:
        FuUnicodeCodepointCaseConvert := 301;
        RETURN;
    301:
        FuUnicodeCodepointCaseConvert := 300;
        RETURN;
    302:
        FuUnicodeCodepointCaseConvert := 303;
        RETURN;
    303:
        FuUnicodeCodepointCaseConvert := 302;
        RETURN;
    304:
        FuUnicodeCodepointCaseConvert := 105;
        RETURN;
    305:
        FuUnicodeCodepointCaseConvert := 73;
        RETURN;
    306:
        FuUnicodeCodepointCaseConvert := 307;
        RETURN;
    307:
        FuUnicodeCodepointCaseConvert := 306;
        RETURN;
    308:
        FuUnicodeCodepointCaseConvert := 309;
        RETURN;
    309:
        FuUnicodeCodepointCaseConvert := 308;
        RETURN;
    310:
        FuUnicodeCodepointCaseConvert := 311;
        RETURN;
    311:
        FuUnicodeCodepointCaseConvert := 310;
        RETURN;
    313:
        FuUnicodeCodepointCaseConvert := 314;
        RETURN;
    314:
        FuUnicodeCodepointCaseConvert := 313;
        RETURN;
    315:
        FuUnicodeCodepointCaseConvert := 316;
        RETURN;
    316:
        FuUnicodeCodepointCaseConvert := 315;
        RETURN;
    317:
        FuUnicodeCodepointCaseConvert := 318;
        RETURN;
    318:
        FuUnicodeCodepointCaseConvert := 317;
        RETURN;
    319:
        FuUnicodeCodepointCaseConvert := 320;
        RETURN;
    320:
        FuUnicodeCodepointCaseConvert := 319;
        RETURN;
    321:
        FuUnicodeCodepointCaseConvert := 322;
        RETURN;
    322:
        FuUnicodeCodepointCaseConvert := 321;
        RETURN;
    323:
        FuUnicodeCodepointCaseConvert := 324;
        RETURN;
    324:
        FuUnicodeCodepointCaseConvert := 323;
        RETURN;
    325:
        FuUnicodeCodepointCaseConvert := 326;
        RETURN;
    326:
        FuUnicodeCodepointCaseConvert := 325;
        RETURN;
    327:
        FuUnicodeCodepointCaseConvert := 328;
        RETURN;
    328:
        FuUnicodeCodepointCaseConvert := 327;
        RETURN;
    330:
        FuUnicodeCodepointCaseConvert := 331;
        RETURN;
    331:
        FuUnicodeCodepointCaseConvert := 330;
        RETURN;
    332:
        FuUnicodeCodepointCaseConvert := 333;
        RETURN;
    333:
        FuUnicodeCodepointCaseConvert := 332;
        RETURN;
    334:
        FuUnicodeCodepointCaseConvert := 335;
        RETURN;
    335:
        FuUnicodeCodepointCaseConvert := 334;
        RETURN;
    336:
        FuUnicodeCodepointCaseConvert := 337;
        RETURN;
    337:
        FuUnicodeCodepointCaseConvert := 336;
        RETURN;
    338:
        FuUnicodeCodepointCaseConvert := 339;
        RETURN;
    339:
        FuUnicodeCodepointCaseConvert := 338;
        RETURN;
    340:
        FuUnicodeCodepointCaseConvert := 341;
        RETURN;
    341:
        FuUnicodeCodepointCaseConvert := 340;
        RETURN;
    342:
        FuUnicodeCodepointCaseConvert := 343;
        RETURN;
    343:
        FuUnicodeCodepointCaseConvert := 342;
        RETURN;
    344:
        FuUnicodeCodepointCaseConvert := 345;
        RETURN;
    345:
        FuUnicodeCodepointCaseConvert := 344;
        RETURN;
    346:
        FuUnicodeCodepointCaseConvert := 347;
        RETURN;
    347:
        FuUnicodeCodepointCaseConvert := 346;
        RETURN;
    348:
        FuUnicodeCodepointCaseConvert := 349;
        RETURN;
    349:
        FuUnicodeCodepointCaseConvert := 348;
        RETURN;
    350:
        FuUnicodeCodepointCaseConvert := 351;
        RETURN;
    351:
        FuUnicodeCodepointCaseConvert := 350;
        RETURN;
    352:
        FuUnicodeCodepointCaseConvert := 353;
        RETURN;
    353:
        FuUnicodeCodepointCaseConvert := 352;
        RETURN;
    354:
        FuUnicodeCodepointCaseConvert := 355;
        RETURN;
    355:
        FuUnicodeCodepointCaseConvert := 354;
        RETURN;
    356:
        FuUnicodeCodepointCaseConvert := 357;
        RETURN;
    357:
        FuUnicodeCodepointCaseConvert := 356;
        RETURN;
    358:
        FuUnicodeCodepointCaseConvert := 359;
        RETURN;
    359:
        FuUnicodeCodepointCaseConvert := 358;
        RETURN;
    360:
        FuUnicodeCodepointCaseConvert := 361;
        RETURN;
    361:
        FuUnicodeCodepointCaseConvert := 360;
        RETURN;
    362:
        FuUnicodeCodepointCaseConvert := 363;
        RETURN;
    363:
        FuUnicodeCodepointCaseConvert := 362;
        RETURN;
    364:
        FuUnicodeCodepointCaseConvert := 365;
        RETURN;
    365:
        FuUnicodeCodepointCaseConvert := 364;
        RETURN;
    366:
        FuUnicodeCodepointCaseConvert := 367;
        RETURN;
    367:
        FuUnicodeCodepointCaseConvert := 366;
        RETURN;
    368:
        FuUnicodeCodepointCaseConvert := 369;
        RETURN;
    369:
        FuUnicodeCodepointCaseConvert := 368;
        RETURN;
    370:
        FuUnicodeCodepointCaseConvert := 371;
        RETURN;
    371:
        FuUnicodeCodepointCaseConvert := 370;
        RETURN;
    372:
        FuUnicodeCodepointCaseConvert := 373;
        RETURN;
    373:
        FuUnicodeCodepointCaseConvert := 372;
        RETURN;
    374:
        FuUnicodeCodepointCaseConvert := 375;
        RETURN;
    375:
        FuUnicodeCodepointCaseConvert := 374;
        RETURN;
    376:
        FuUnicodeCodepointCaseConvert := 255;
        RETURN;
    377:
        FuUnicodeCodepointCaseConvert := 378;
        RETURN;
    378:
        FuUnicodeCodepointCaseConvert := 377;
        RETURN;
    379:
        FuUnicodeCodepointCaseConvert := 380;
        RETURN;
    380:
        FuUnicodeCodepointCaseConvert := 379;
        RETURN;
    381:
        FuUnicodeCodepointCaseConvert := 382;
        RETURN;
    382:
        FuUnicodeCodepointCaseConvert := 381;
        RETURN;
    383:
        FuUnicodeCodepointCaseConvert := 83;
        RETURN;
    384:
        FuUnicodeCodepointCaseConvert := 579;
        RETURN;
    385:
        FuUnicodeCodepointCaseConvert := 595;
        RETURN;
    386:
        FuUnicodeCodepointCaseConvert := 387;
        RETURN;
    387:
        FuUnicodeCodepointCaseConvert := 386;
        RETURN;
    388:
        FuUnicodeCodepointCaseConvert := 389;
        RETURN;
    389:
        FuUnicodeCodepointCaseConvert := 388;
        RETURN;
    390:
        FuUnicodeCodepointCaseConvert := 596;
        RETURN;
    391:
        FuUnicodeCodepointCaseConvert := 392;
        RETURN;
    392:
        FuUnicodeCodepointCaseConvert := 391;
        RETURN;
    393:
        FuUnicodeCodepointCaseConvert := 598;
        RETURN;
    394:
        FuUnicodeCodepointCaseConvert := 599;
        RETURN;
    395:
        FuUnicodeCodepointCaseConvert := 396;
        RETURN;
    396:
        FuUnicodeCodepointCaseConvert := 395;
        RETURN;
    398:
        FuUnicodeCodepointCaseConvert := 477;
        RETURN;
    399:
        FuUnicodeCodepointCaseConvert := 601;
        RETURN;
    400:
        FuUnicodeCodepointCaseConvert := 603;
        RETURN;
    401:
        FuUnicodeCodepointCaseConvert := 402;
        RETURN;
    402:
        FuUnicodeCodepointCaseConvert := 401;
        RETURN;
    403:
        FuUnicodeCodepointCaseConvert := 608;
        RETURN;
    404:
        FuUnicodeCodepointCaseConvert := 611;
        RETURN;
    405:
        FuUnicodeCodepointCaseConvert := 502;
        RETURN;
    406:
        FuUnicodeCodepointCaseConvert := 617;
        RETURN;
    407:
        FuUnicodeCodepointCaseConvert := 616;
        RETURN;
    408:
        FuUnicodeCodepointCaseConvert := 409;
        RETURN;
    409:
        FuUnicodeCodepointCaseConvert := 408;
        RETURN;
    410:
        FuUnicodeCodepointCaseConvert := 573;
        RETURN;
    412:
        FuUnicodeCodepointCaseConvert := 623;
        RETURN;
    413:
        FuUnicodeCodepointCaseConvert := 626;
        RETURN;
    414:
        FuUnicodeCodepointCaseConvert := 544;
        RETURN;
    415:
        FuUnicodeCodepointCaseConvert := 629;
        RETURN;
    416:
        FuUnicodeCodepointCaseConvert := 417;
        RETURN;
    417:
        FuUnicodeCodepointCaseConvert := 416;
        RETURN;
    418:
        FuUnicodeCodepointCaseConvert := 419;
        RETURN;
    419:
        FuUnicodeCodepointCaseConvert := 418;
        RETURN;
    420:
        FuUnicodeCodepointCaseConvert := 421;
        RETURN;
    421:
        FuUnicodeCodepointCaseConvert := 420;
        RETURN;
    422:
        FuUnicodeCodepointCaseConvert := 640;
        RETURN;
    423:
        FuUnicodeCodepointCaseConvert := 424;
        RETURN;
    424:
        FuUnicodeCodepointCaseConvert := 423;
        RETURN;
    425:
        FuUnicodeCodepointCaseConvert := 643;
        RETURN;
    428:
        FuUnicodeCodepointCaseConvert := 429;
        RETURN;
    429:
        FuUnicodeCodepointCaseConvert := 428;
        RETURN;
    430:
        FuUnicodeCodepointCaseConvert := 648;
        RETURN;
    431:
        FuUnicodeCodepointCaseConvert := 432;
        RETURN;
    432:
        FuUnicodeCodepointCaseConvert := 431;
        RETURN;
    433:
        FuUnicodeCodepointCaseConvert := 650;
        RETURN;
    434:
        FuUnicodeCodepointCaseConvert := 651;
        RETURN;
    435:
        FuUnicodeCodepointCaseConvert := 436;
        RETURN;
    436:
        FuUnicodeCodepointCaseConvert := 435;
        RETURN;
    437:
        FuUnicodeCodepointCaseConvert := 438;
        RETURN;
    438:
        FuUnicodeCodepointCaseConvert := 437;
        RETURN;
    439:
        FuUnicodeCodepointCaseConvert := 658;
        RETURN;
    440:
        FuUnicodeCodepointCaseConvert := 441;
        RETURN;
    441:
        FuUnicodeCodepointCaseConvert := 440;
        RETURN;
    444:
        FuUnicodeCodepointCaseConvert := 445;
        RETURN;
    445:
        FuUnicodeCodepointCaseConvert := 444;
        RETURN;
    447:
        FuUnicodeCodepointCaseConvert := 503;
        RETURN;
    452:
        FuUnicodeCodepointCaseConvert := 453;
        RETURN;
    453:
        FuUnicodeCodepointCaseConvert := 453;
        RETURN;
    454:
        FuUnicodeCodepointCaseConvert := 453;
        RETURN;
    455:
        FuUnicodeCodepointCaseConvert := 456;
        RETURN;
    456:
        FuUnicodeCodepointCaseConvert := 456;
        RETURN;
    457:
        FuUnicodeCodepointCaseConvert := 456;
        RETURN;
    458:
        FuUnicodeCodepointCaseConvert := 459;
        RETURN;
    459:
        FuUnicodeCodepointCaseConvert := 459;
        RETURN;
    460:
        FuUnicodeCodepointCaseConvert := 459;
        RETURN;
    461:
        FuUnicodeCodepointCaseConvert := 462;
        RETURN;
    462:
        FuUnicodeCodepointCaseConvert := 461;
        RETURN;
    463:
        FuUnicodeCodepointCaseConvert := 464;
        RETURN;
    464:
        FuUnicodeCodepointCaseConvert := 463;
        RETURN;
    465:
        FuUnicodeCodepointCaseConvert := 466;
        RETURN;
    466:
        FuUnicodeCodepointCaseConvert := 465;
        RETURN;
    467:
        FuUnicodeCodepointCaseConvert := 468;
        RETURN;
    468:
        FuUnicodeCodepointCaseConvert := 467;
        RETURN;
    469:
        FuUnicodeCodepointCaseConvert := 470;
        RETURN;
    470:
        FuUnicodeCodepointCaseConvert := 469;
        RETURN;
    471:
        FuUnicodeCodepointCaseConvert := 472;
        RETURN;
    472:
        FuUnicodeCodepointCaseConvert := 471;
        RETURN;
    473:
        FuUnicodeCodepointCaseConvert := 474;
        RETURN;
    474:
        FuUnicodeCodepointCaseConvert := 473;
        RETURN;
    475:
        FuUnicodeCodepointCaseConvert := 476;
        RETURN;
    476:
        FuUnicodeCodepointCaseConvert := 475;
        RETURN;
    477:
        FuUnicodeCodepointCaseConvert := 398;
        RETURN;
    478:
        FuUnicodeCodepointCaseConvert := 479;
        RETURN;
    479:
        FuUnicodeCodepointCaseConvert := 478;
        RETURN;
    480:
        FuUnicodeCodepointCaseConvert := 481;
        RETURN;
    481:
        FuUnicodeCodepointCaseConvert := 480;
        RETURN;
    482:
        FuUnicodeCodepointCaseConvert := 483;
        RETURN;
    483:
        FuUnicodeCodepointCaseConvert := 482;
        RETURN;
    484:
        FuUnicodeCodepointCaseConvert := 485;
        RETURN;
    485:
        FuUnicodeCodepointCaseConvert := 484;
        RETURN;
    486:
        FuUnicodeCodepointCaseConvert := 487;
        RETURN;
    487:
        FuUnicodeCodepointCaseConvert := 486;
        RETURN;
    488:
        FuUnicodeCodepointCaseConvert := 489;
        RETURN;
    489:
        FuUnicodeCodepointCaseConvert := 488;
        RETURN;
    490:
        FuUnicodeCodepointCaseConvert := 491;
        RETURN;
    491:
        FuUnicodeCodepointCaseConvert := 490;
        RETURN;
    492:
        FuUnicodeCodepointCaseConvert := 493;
        RETURN;
    493:
        FuUnicodeCodepointCaseConvert := 492;
        RETURN;
    494:
        FuUnicodeCodepointCaseConvert := 495;
        RETURN;
    495:
        FuUnicodeCodepointCaseConvert := 494;
        RETURN;
    497:
        FuUnicodeCodepointCaseConvert := 498;
        RETURN;
    498:
        FuUnicodeCodepointCaseConvert := 498;
        RETURN;
    499:
        FuUnicodeCodepointCaseConvert := 498;
        RETURN;
    500:
        FuUnicodeCodepointCaseConvert := 501;
        RETURN;
    501:
        FuUnicodeCodepointCaseConvert := 500;
        RETURN;
    502:
        FuUnicodeCodepointCaseConvert := 405;
        RETURN;
    503:
        FuUnicodeCodepointCaseConvert := 447;
        RETURN;
    504:
        FuUnicodeCodepointCaseConvert := 505;
        RETURN;
    505:
        FuUnicodeCodepointCaseConvert := 504;
        RETURN;
    506:
        FuUnicodeCodepointCaseConvert := 507;
        RETURN;
    507:
        FuUnicodeCodepointCaseConvert := 506;
        RETURN;
    508:
        FuUnicodeCodepointCaseConvert := 509;
        RETURN;
    509:
        FuUnicodeCodepointCaseConvert := 508;
        RETURN;
    510:
        FuUnicodeCodepointCaseConvert := 511;
        RETURN;
    511:
        FuUnicodeCodepointCaseConvert := 510;
        RETURN;
    512:
        FuUnicodeCodepointCaseConvert := 513;
        RETURN;
    513:
        FuUnicodeCodepointCaseConvert := 512;
        RETURN;
    514:
        FuUnicodeCodepointCaseConvert := 515;
        RETURN;
    515:
        FuUnicodeCodepointCaseConvert := 514;
        RETURN;
    516:
        FuUnicodeCodepointCaseConvert := 517;
        RETURN;
    517:
        FuUnicodeCodepointCaseConvert := 516;
        RETURN;
    518:
        FuUnicodeCodepointCaseConvert := 519;
        RETURN;
    519:
        FuUnicodeCodepointCaseConvert := 518;
        RETURN;
    520:
        FuUnicodeCodepointCaseConvert := 521;
        RETURN;
    521:
        FuUnicodeCodepointCaseConvert := 520;
        RETURN;
    522:
        FuUnicodeCodepointCaseConvert := 523;
        RETURN;
    523:
        FuUnicodeCodepointCaseConvert := 522;
        RETURN;
    524:
        FuUnicodeCodepointCaseConvert := 525;
        RETURN;
    525:
        FuUnicodeCodepointCaseConvert := 524;
        RETURN;
    526:
        FuUnicodeCodepointCaseConvert := 527;
        RETURN;
    527:
        FuUnicodeCodepointCaseConvert := 526;
        RETURN;
    528:
        FuUnicodeCodepointCaseConvert := 529;
        RETURN;
    529:
        FuUnicodeCodepointCaseConvert := 528;
        RETURN;
    530:
        FuUnicodeCodepointCaseConvert := 531;
        RETURN;
    531:
        FuUnicodeCodepointCaseConvert := 530;
        RETURN;
    532:
        FuUnicodeCodepointCaseConvert := 533;
        RETURN;
    533:
        FuUnicodeCodepointCaseConvert := 532;
        RETURN;
    534:
        FuUnicodeCodepointCaseConvert := 535;
        RETURN;
    535:
        FuUnicodeCodepointCaseConvert := 534;
        RETURN;
    536:
        FuUnicodeCodepointCaseConvert := 537;
        RETURN;
    537:
        FuUnicodeCodepointCaseConvert := 536;
        RETURN;
    538:
        FuUnicodeCodepointCaseConvert := 539;
        RETURN;
    539:
        FuUnicodeCodepointCaseConvert := 538;
        RETURN;
    540:
        FuUnicodeCodepointCaseConvert := 541;
        RETURN;
    541:
        FuUnicodeCodepointCaseConvert := 540;
        RETURN;
    542:
        FuUnicodeCodepointCaseConvert := 543;
        RETURN;
    543:
        FuUnicodeCodepointCaseConvert := 542;
        RETURN;
    544:
        FuUnicodeCodepointCaseConvert := 414;
        RETURN;
    546:
        FuUnicodeCodepointCaseConvert := 547;
        RETURN;
    547:
        FuUnicodeCodepointCaseConvert := 546;
        RETURN;
    548:
        FuUnicodeCodepointCaseConvert := 549;
        RETURN;
    549:
        FuUnicodeCodepointCaseConvert := 548;
        RETURN;
    550:
        FuUnicodeCodepointCaseConvert := 551;
        RETURN;
    551:
        FuUnicodeCodepointCaseConvert := 550;
        RETURN;
    552:
        FuUnicodeCodepointCaseConvert := 553;
        RETURN;
    553:
        FuUnicodeCodepointCaseConvert := 552;
        RETURN;
    554:
        FuUnicodeCodepointCaseConvert := 555;
        RETURN;
    555:
        FuUnicodeCodepointCaseConvert := 554;
        RETURN;
    556:
        FuUnicodeCodepointCaseConvert := 557;
        RETURN;
    557:
        FuUnicodeCodepointCaseConvert := 556;
        RETURN;
    558:
        FuUnicodeCodepointCaseConvert := 559;
        RETURN;
    559:
        FuUnicodeCodepointCaseConvert := 558;
        RETURN;
    560:
        FuUnicodeCodepointCaseConvert := 561;
        RETURN;
    561:
        FuUnicodeCodepointCaseConvert := 560;
        RETURN;
    562:
        FuUnicodeCodepointCaseConvert := 563;
        RETURN;
    563:
        FuUnicodeCodepointCaseConvert := 562;
        RETURN;
    570:
        FuUnicodeCodepointCaseConvert := 11365;
        RETURN;
    571:
        FuUnicodeCodepointCaseConvert := 572;
        RETURN;
    572:
        FuUnicodeCodepointCaseConvert := 571;
        RETURN;
    573:
        FuUnicodeCodepointCaseConvert := 410;
        RETURN;
    574:
        FuUnicodeCodepointCaseConvert := 11366;
        RETURN;
    575:
        FuUnicodeCodepointCaseConvert := 11390;
        RETURN;
    576:
        FuUnicodeCodepointCaseConvert := 11391;
        RETURN;
    577:
        FuUnicodeCodepointCaseConvert := 578;
        RETURN;
    578:
        FuUnicodeCodepointCaseConvert := 577;
        RETURN;
    579:
        FuUnicodeCodepointCaseConvert := 384;
        RETURN;
    580:
        FuUnicodeCodepointCaseConvert := 649;
        RETURN;
    581:
        FuUnicodeCodepointCaseConvert := 652;
        RETURN;
    582:
        FuUnicodeCodepointCaseConvert := 583;
        RETURN;
    583:
        FuUnicodeCodepointCaseConvert := 582;
        RETURN;
    584:
        FuUnicodeCodepointCaseConvert := 585;
        RETURN;
    585:
        FuUnicodeCodepointCaseConvert := 584;
        RETURN;
    586:
        FuUnicodeCodepointCaseConvert := 587;
        RETURN;
    587:
        FuUnicodeCodepointCaseConvert := 586;
        RETURN;
    588:
        FuUnicodeCodepointCaseConvert := 589;
        RETURN;
    589:
        FuUnicodeCodepointCaseConvert := 588;
        RETURN;
    590:
        FuUnicodeCodepointCaseConvert := 591;
        RETURN;
    591:
        FuUnicodeCodepointCaseConvert := 590;
        RETURN;
    592:
        FuUnicodeCodepointCaseConvert := 11375;
        RETURN;
    593:
        FuUnicodeCodepointCaseConvert := 11373;
        RETURN;
    594:
        FuUnicodeCodepointCaseConvert := 11376;
        RETURN;
    595:
        FuUnicodeCodepointCaseConvert := 385;
        RETURN;
    596:
        FuUnicodeCodepointCaseConvert := 390;
        RETURN;
    598:
        FuUnicodeCodepointCaseConvert := 393;
        RETURN;
    599:
        FuUnicodeCodepointCaseConvert := 394;
        RETURN;
    601:
        FuUnicodeCodepointCaseConvert := 399;
        RETURN;
    603:
        FuUnicodeCodepointCaseConvert := 400;
        RETURN;
    604:
        FuUnicodeCodepointCaseConvert := 42923;
        RETURN;
    608:
        FuUnicodeCodepointCaseConvert := 403;
        RETURN;
    609:
        FuUnicodeCodepointCaseConvert := 42924;
        RETURN;
    611:
        FuUnicodeCodepointCaseConvert := 404;
        RETURN;
    613:
        FuUnicodeCodepointCaseConvert := 42893;
        RETURN;
    614:
        FuUnicodeCodepointCaseConvert := 42922;
        RETURN;
    616:
        FuUnicodeCodepointCaseConvert := 407;
        RETURN;
    617:
        FuUnicodeCodepointCaseConvert := 406;
        RETURN;
    618:
        FuUnicodeCodepointCaseConvert := 42926;
        RETURN;
    619:
        FuUnicodeCodepointCaseConvert := 11362;
        RETURN;
    620:
        FuUnicodeCodepointCaseConvert := 42925;
        RETURN;
    623:
        FuUnicodeCodepointCaseConvert := 412;
        RETURN;
    625:
        FuUnicodeCodepointCaseConvert := 11374;
        RETURN;
    626:
        FuUnicodeCodepointCaseConvert := 413;
        RETURN;
    629:
        FuUnicodeCodepointCaseConvert := 415;
        RETURN;
    637:
        FuUnicodeCodepointCaseConvert := 11364;
        RETURN;
    640:
        FuUnicodeCodepointCaseConvert := 422;
        RETURN;
    642:
        FuUnicodeCodepointCaseConvert := 42949;
        RETURN;
    643:
        FuUnicodeCodepointCaseConvert := 425;
        RETURN;
    647:
        FuUnicodeCodepointCaseConvert := 42929;
        RETURN;
    648:
        FuUnicodeCodepointCaseConvert := 430;
        RETURN;
    649:
        FuUnicodeCodepointCaseConvert := 580;
        RETURN;
    650:
        FuUnicodeCodepointCaseConvert := 433;
        RETURN;
    651:
        FuUnicodeCodepointCaseConvert := 434;
        RETURN;
    652:
        FuUnicodeCodepointCaseConvert := 581;
        RETURN;
    658:
        FuUnicodeCodepointCaseConvert := 439;
        RETURN;
    669:
        FuUnicodeCodepointCaseConvert := 42930;
        RETURN;
    670:
        FuUnicodeCodepointCaseConvert := 42928;
        RETURN;
    837:
        FuUnicodeCodepointCaseConvert := 921;
        RETURN;
    880:
        FuUnicodeCodepointCaseConvert := 881;
        RETURN;
    881:
        FuUnicodeCodepointCaseConvert := 880;
        RETURN;
    882:
        FuUnicodeCodepointCaseConvert := 883;
        RETURN;
    883:
        FuUnicodeCodepointCaseConvert := 882;
        RETURN;
    886:
        FuUnicodeCodepointCaseConvert := 887;
        RETURN;
    887:
        FuUnicodeCodepointCaseConvert := 886;
        RETURN;
    891:
        FuUnicodeCodepointCaseConvert := 1021;
        RETURN;
    892:
        FuUnicodeCodepointCaseConvert := 1022;
        RETURN;
    893:
        FuUnicodeCodepointCaseConvert := 1023;
        RETURN;
    895:
        FuUnicodeCodepointCaseConvert := 1011;
        RETURN;
    902:
        FuUnicodeCodepointCaseConvert := 940;
        RETURN;
    904:
        FuUnicodeCodepointCaseConvert := 941;
        RETURN;
    905:
        FuUnicodeCodepointCaseConvert := 942;
        RETURN;
    906:
        FuUnicodeCodepointCaseConvert := 943;
        RETURN;
    908:
        FuUnicodeCodepointCaseConvert := 972;
        RETURN;
    910:
        FuUnicodeCodepointCaseConvert := 973;
        RETURN;
    911:
        FuUnicodeCodepointCaseConvert := 974;
        RETURN;
    913:
        FuUnicodeCodepointCaseConvert := 945;
        RETURN;
    914:
        FuUnicodeCodepointCaseConvert := 946;
        RETURN;
    915:
        FuUnicodeCodepointCaseConvert := 947;
        RETURN;
    916:
        FuUnicodeCodepointCaseConvert := 948;
        RETURN;
    917:
        FuUnicodeCodepointCaseConvert := 949;
        RETURN;
    918:
        FuUnicodeCodepointCaseConvert := 950;
        RETURN;
    919:
        FuUnicodeCodepointCaseConvert := 951;
        RETURN;
    920:
        FuUnicodeCodepointCaseConvert := 952;
        RETURN;
    921:
        FuUnicodeCodepointCaseConvert := 953;
        RETURN;
    922:
        FuUnicodeCodepointCaseConvert := 954;
        RETURN;
    923:
        FuUnicodeCodepointCaseConvert := 955;
        RETURN;
    924:
        FuUnicodeCodepointCaseConvert := 956;
        RETURN;
    925:
        FuUnicodeCodepointCaseConvert := 957;
        RETURN;
    926:
        FuUnicodeCodepointCaseConvert := 958;
        RETURN;
    927:
        FuUnicodeCodepointCaseConvert := 959;
        RETURN;
    928:
        FuUnicodeCodepointCaseConvert := 960;
        RETURN;
    929:
        FuUnicodeCodepointCaseConvert := 961;
        RETURN;
    931:
        FuUnicodeCodepointCaseConvert := 963;
        RETURN;
    932:
        FuUnicodeCodepointCaseConvert := 964;
        RETURN;
    933:
        FuUnicodeCodepointCaseConvert := 965;
        RETURN;
    934:
        FuUnicodeCodepointCaseConvert := 966;
        RETURN;
    935:
        FuUnicodeCodepointCaseConvert := 967;
        RETURN;
    936:
        FuUnicodeCodepointCaseConvert := 968;
        RETURN;
    937:
        FuUnicodeCodepointCaseConvert := 969;
        RETURN;
    938:
        FuUnicodeCodepointCaseConvert := 970;
        RETURN;
    939:
        FuUnicodeCodepointCaseConvert := 971;
        RETURN;
    940:
        FuUnicodeCodepointCaseConvert := 902;
        RETURN;
    941:
        FuUnicodeCodepointCaseConvert := 904;
        RETURN;
    942:
        FuUnicodeCodepointCaseConvert := 905;
        RETURN;
    943:
        FuUnicodeCodepointCaseConvert := 906;
        RETURN;
    945:
        FuUnicodeCodepointCaseConvert := 913;
        RETURN;
    946:
        FuUnicodeCodepointCaseConvert := 914;
        RETURN;
    947:
        FuUnicodeCodepointCaseConvert := 915;
        RETURN;
    948:
        FuUnicodeCodepointCaseConvert := 916;
        RETURN;
    949:
        FuUnicodeCodepointCaseConvert := 917;
        RETURN;
    950:
        FuUnicodeCodepointCaseConvert := 918;
        RETURN;
    951:
        FuUnicodeCodepointCaseConvert := 919;
        RETURN;
    952:
        FuUnicodeCodepointCaseConvert := 920;
        RETURN;
    953:
        FuUnicodeCodepointCaseConvert := 921;
        RETURN;
    954:
        FuUnicodeCodepointCaseConvert := 922;
        RETURN;
    955:
        FuUnicodeCodepointCaseConvert := 923;
        RETURN;
    956:
        FuUnicodeCodepointCaseConvert := 924;
        RETURN;
    957:
        FuUnicodeCodepointCaseConvert := 925;
        RETURN;
    958:
        FuUnicodeCodepointCaseConvert := 926;
        RETURN;
    959:
        FuUnicodeCodepointCaseConvert := 927;
        RETURN;
    960:
        FuUnicodeCodepointCaseConvert := 928;
        RETURN;
    961:
        FuUnicodeCodepointCaseConvert := 929;
        RETURN;
    962:
        FuUnicodeCodepointCaseConvert := 931;
        RETURN;
    963:
        FuUnicodeCodepointCaseConvert := 931;
        RETURN;
    964:
        FuUnicodeCodepointCaseConvert := 932;
        RETURN;
    965:
        FuUnicodeCodepointCaseConvert := 933;
        RETURN;
    966:
        FuUnicodeCodepointCaseConvert := 934;
        RETURN;
    967:
        FuUnicodeCodepointCaseConvert := 935;
        RETURN;
    968:
        FuUnicodeCodepointCaseConvert := 936;
        RETURN;
    969:
        FuUnicodeCodepointCaseConvert := 937;
        RETURN;
    970:
        FuUnicodeCodepointCaseConvert := 938;
        RETURN;
    971:
        FuUnicodeCodepointCaseConvert := 939;
        RETURN;
    972:
        FuUnicodeCodepointCaseConvert := 908;
        RETURN;
    973:
        FuUnicodeCodepointCaseConvert := 910;
        RETURN;
    974:
        FuUnicodeCodepointCaseConvert := 911;
        RETURN;
    975:
        FuUnicodeCodepointCaseConvert := 983;
        RETURN;
    976:
        FuUnicodeCodepointCaseConvert := 914;
        RETURN;
    977:
        FuUnicodeCodepointCaseConvert := 920;
        RETURN;
    981:
        FuUnicodeCodepointCaseConvert := 934;
        RETURN;
    982:
        FuUnicodeCodepointCaseConvert := 928;
        RETURN;
    983:
        FuUnicodeCodepointCaseConvert := 975;
        RETURN;
    984:
        FuUnicodeCodepointCaseConvert := 985;
        RETURN;
    985:
        FuUnicodeCodepointCaseConvert := 984;
        RETURN;
    986:
        FuUnicodeCodepointCaseConvert := 987;
        RETURN;
    987:
        FuUnicodeCodepointCaseConvert := 986;
        RETURN;
    988:
        FuUnicodeCodepointCaseConvert := 989;
        RETURN;
    989:
        FuUnicodeCodepointCaseConvert := 988;
        RETURN;
    990:
        FuUnicodeCodepointCaseConvert := 991;
        RETURN;
    991:
        FuUnicodeCodepointCaseConvert := 990;
        RETURN;
    992:
        FuUnicodeCodepointCaseConvert := 993;
        RETURN;
    993:
        FuUnicodeCodepointCaseConvert := 992;
        RETURN;
    994:
        FuUnicodeCodepointCaseConvert := 995;
        RETURN;
    995:
        FuUnicodeCodepointCaseConvert := 994;
        RETURN;
    996:
        FuUnicodeCodepointCaseConvert := 997;
        RETURN;
    997:
        FuUnicodeCodepointCaseConvert := 996;
        RETURN;
    998:
        FuUnicodeCodepointCaseConvert := 999;
        RETURN;
    999:
        FuUnicodeCodepointCaseConvert := 998;
        RETURN;
    1000:
        FuUnicodeCodepointCaseConvert := 1001;
        RETURN;
    1001:
        FuUnicodeCodepointCaseConvert := 1000;
        RETURN;
    1002:
        FuUnicodeCodepointCaseConvert := 1003;
        RETURN;
    1003:
        FuUnicodeCodepointCaseConvert := 1002;
        RETURN;
    1004:
        FuUnicodeCodepointCaseConvert := 1005;
        RETURN;
    1005:
        FuUnicodeCodepointCaseConvert := 1004;
        RETURN;
    1006:
        FuUnicodeCodepointCaseConvert := 1007;
        RETURN;
    1007:
        FuUnicodeCodepointCaseConvert := 1006;
        RETURN;
    1008:
        FuUnicodeCodepointCaseConvert := 922;
        RETURN;
    1009:
        FuUnicodeCodepointCaseConvert := 929;
        RETURN;
    1010:
        FuUnicodeCodepointCaseConvert := 1017;
        RETURN;
    1011:
        FuUnicodeCodepointCaseConvert := 895;
        RETURN;
    1012:
        FuUnicodeCodepointCaseConvert := 952;
        RETURN;
    1013:
        FuUnicodeCodepointCaseConvert := 917;
        RETURN;
    1015:
        FuUnicodeCodepointCaseConvert := 1016;
        RETURN;
    1016:
        FuUnicodeCodepointCaseConvert := 1015;
        RETURN;
    1017:
        FuUnicodeCodepointCaseConvert := 1010;
        RETURN;
    1018:
        FuUnicodeCodepointCaseConvert := 1019;
        RETURN;
    1019:
        FuUnicodeCodepointCaseConvert := 1018;
        RETURN;
    1021:
        FuUnicodeCodepointCaseConvert := 891;
        RETURN;
    1022:
        FuUnicodeCodepointCaseConvert := 892;
        RETURN;
    1023:
        FuUnicodeCodepointCaseConvert := 893;
        RETURN;
    1024:
        FuUnicodeCodepointCaseConvert := 1104;
        RETURN;
    1025:
        FuUnicodeCodepointCaseConvert := 1105;
        RETURN;
    1026:
        FuUnicodeCodepointCaseConvert := 1106;
        RETURN;
    1027:
        FuUnicodeCodepointCaseConvert := 1107;
        RETURN;
    1028:
        FuUnicodeCodepointCaseConvert := 1108;
        RETURN;
    1029:
        FuUnicodeCodepointCaseConvert := 1109;
        RETURN;
    1030:
        FuUnicodeCodepointCaseConvert := 1110;
        RETURN;
    1031:
        FuUnicodeCodepointCaseConvert := 1111;
        RETURN;
    1032:
        FuUnicodeCodepointCaseConvert := 1112;
        RETURN;
    1033:
        FuUnicodeCodepointCaseConvert := 1113;
        RETURN;
    1034:
        FuUnicodeCodepointCaseConvert := 1114;
        RETURN;
    1035:
        FuUnicodeCodepointCaseConvert := 1115;
        RETURN;
    1036:
        FuUnicodeCodepointCaseConvert := 1116;
        RETURN;
    1037:
        FuUnicodeCodepointCaseConvert := 1117;
        RETURN;
    1038:
        FuUnicodeCodepointCaseConvert := 1118;
        RETURN;
    1039:
        FuUnicodeCodepointCaseConvert := 1119;
        RETURN;
    1040:
        FuUnicodeCodepointCaseConvert := 1072;
        RETURN;
    1041:
        FuUnicodeCodepointCaseConvert := 1073;
        RETURN;
    1042:
        FuUnicodeCodepointCaseConvert := 1074;
        RETURN;
    1043:
        FuUnicodeCodepointCaseConvert := 1075;
        RETURN;
    1044:
        FuUnicodeCodepointCaseConvert := 1076;
        RETURN;
    1045:
        FuUnicodeCodepointCaseConvert := 1077;
        RETURN;
    1046:
        FuUnicodeCodepointCaseConvert := 1078;
        RETURN;
    1047:
        FuUnicodeCodepointCaseConvert := 1079;
        RETURN;
    1048:
        FuUnicodeCodepointCaseConvert := 1080;
        RETURN;
    1049:
        FuUnicodeCodepointCaseConvert := 1081;
        RETURN;
    1050:
        FuUnicodeCodepointCaseConvert := 1082;
        RETURN;
    1051:
        FuUnicodeCodepointCaseConvert := 1083;
        RETURN;
    1052:
        FuUnicodeCodepointCaseConvert := 1084;
        RETURN;
    1053:
        FuUnicodeCodepointCaseConvert := 1085;
        RETURN;
    1054:
        FuUnicodeCodepointCaseConvert := 1086;
        RETURN;
    1055:
        FuUnicodeCodepointCaseConvert := 1087;
        RETURN;
    1056:
        FuUnicodeCodepointCaseConvert := 1088;
        RETURN;
    1057:
        FuUnicodeCodepointCaseConvert := 1089;
        RETURN;
    1058:
        FuUnicodeCodepointCaseConvert := 1090;
        RETURN;
    1059:
        FuUnicodeCodepointCaseConvert := 1091;
        RETURN;
    1060:
        FuUnicodeCodepointCaseConvert := 1092;
        RETURN;
    1061:
        FuUnicodeCodepointCaseConvert := 1093;
        RETURN;
    1062:
        FuUnicodeCodepointCaseConvert := 1094;
        RETURN;
    1063:
        FuUnicodeCodepointCaseConvert := 1095;
        RETURN;
    1064:
        FuUnicodeCodepointCaseConvert := 1096;
        RETURN;
    1065:
        FuUnicodeCodepointCaseConvert := 1097;
        RETURN;
    1066:
        FuUnicodeCodepointCaseConvert := 1098;
        RETURN;
    1067:
        FuUnicodeCodepointCaseConvert := 1099;
        RETURN;
    1068:
        FuUnicodeCodepointCaseConvert := 1100;
        RETURN;
    1069:
        FuUnicodeCodepointCaseConvert := 1101;
        RETURN;
    1070:
        FuUnicodeCodepointCaseConvert := 1102;
        RETURN;
    1071:
        FuUnicodeCodepointCaseConvert := 1103;
        RETURN;
    1072:
        FuUnicodeCodepointCaseConvert := 1040;
        RETURN;
    1073:
        FuUnicodeCodepointCaseConvert := 1041;
        RETURN;
    1074:
        FuUnicodeCodepointCaseConvert := 1042;
        RETURN;
    1075:
        FuUnicodeCodepointCaseConvert := 1043;
        RETURN;
    1076:
        FuUnicodeCodepointCaseConvert := 1044;
        RETURN;
    1077:
        FuUnicodeCodepointCaseConvert := 1045;
        RETURN;
    1078:
        FuUnicodeCodepointCaseConvert := 1046;
        RETURN;
    1079:
        FuUnicodeCodepointCaseConvert := 1047;
        RETURN;
    1080:
        FuUnicodeCodepointCaseConvert := 1048;
        RETURN;
    1081:
        FuUnicodeCodepointCaseConvert := 1049;
        RETURN;
    1082:
        FuUnicodeCodepointCaseConvert := 1050;
        RETURN;
    1083:
        FuUnicodeCodepointCaseConvert := 1051;
        RETURN;
    1084:
        FuUnicodeCodepointCaseConvert := 1052;
        RETURN;
    1085:
        FuUnicodeCodepointCaseConvert := 1053;
        RETURN;
    1086:
        FuUnicodeCodepointCaseConvert := 1054;
        RETURN;
    1087:
        FuUnicodeCodepointCaseConvert := 1055;
        RETURN;
    1088:
        FuUnicodeCodepointCaseConvert := 1056;
        RETURN;
    1089:
        FuUnicodeCodepointCaseConvert := 1057;
        RETURN;
    1090:
        FuUnicodeCodepointCaseConvert := 1058;
        RETURN;
    1091:
        FuUnicodeCodepointCaseConvert := 1059;
        RETURN;
    1092:
        FuUnicodeCodepointCaseConvert := 1060;
        RETURN;
    1093:
        FuUnicodeCodepointCaseConvert := 1061;
        RETURN;
    1094:
        FuUnicodeCodepointCaseConvert := 1062;
        RETURN;
    1095:
        FuUnicodeCodepointCaseConvert := 1063;
        RETURN;
    1096:
        FuUnicodeCodepointCaseConvert := 1064;
        RETURN;
    1097:
        FuUnicodeCodepointCaseConvert := 1065;
        RETURN;
    1098:
        FuUnicodeCodepointCaseConvert := 1066;
        RETURN;
    1099:
        FuUnicodeCodepointCaseConvert := 1067;
        RETURN;
    1100:
        FuUnicodeCodepointCaseConvert := 1068;
        RETURN;
    1101:
        FuUnicodeCodepointCaseConvert := 1069;
        RETURN;
    1102:
        FuUnicodeCodepointCaseConvert := 1070;
        RETURN;
    1103:
        FuUnicodeCodepointCaseConvert := 1071;
        RETURN;
    1104:
        FuUnicodeCodepointCaseConvert := 1024;
        RETURN;
    1105:
        FuUnicodeCodepointCaseConvert := 1025;
        RETURN;
    1106:
        FuUnicodeCodepointCaseConvert := 1026;
        RETURN;
    1107:
        FuUnicodeCodepointCaseConvert := 1027;
        RETURN;
    1108:
        FuUnicodeCodepointCaseConvert := 1028;
        RETURN;
    1109:
        FuUnicodeCodepointCaseConvert := 1029;
        RETURN;
    1110:
        FuUnicodeCodepointCaseConvert := 1030;
        RETURN;
    1111:
        FuUnicodeCodepointCaseConvert := 1031;
        RETURN;
    1112:
        FuUnicodeCodepointCaseConvert := 1032;
        RETURN;
    1113:
        FuUnicodeCodepointCaseConvert := 1033;
        RETURN;
    1114:
        FuUnicodeCodepointCaseConvert := 1034;
        RETURN;
    1115:
        FuUnicodeCodepointCaseConvert := 1035;
        RETURN;
    1116:
        FuUnicodeCodepointCaseConvert := 1036;
        RETURN;
    1117:
        FuUnicodeCodepointCaseConvert := 1037;
        RETURN;
    1118:
        FuUnicodeCodepointCaseConvert := 1038;
        RETURN;
    1119:
        FuUnicodeCodepointCaseConvert := 1039;
        RETURN;
    1120:
        FuUnicodeCodepointCaseConvert := 1121;
        RETURN;
    1121:
        FuUnicodeCodepointCaseConvert := 1120;
        RETURN;
    1122:
        FuUnicodeCodepointCaseConvert := 1123;
        RETURN;
    1123:
        FuUnicodeCodepointCaseConvert := 1122;
        RETURN;
    1124:
        FuUnicodeCodepointCaseConvert := 1125;
        RETURN;
    1125:
        FuUnicodeCodepointCaseConvert := 1124;
        RETURN;
    1126:
        FuUnicodeCodepointCaseConvert := 1127;
        RETURN;
    1127:
        FuUnicodeCodepointCaseConvert := 1126;
        RETURN;
    1128:
        FuUnicodeCodepointCaseConvert := 1129;
        RETURN;
    1129:
        FuUnicodeCodepointCaseConvert := 1128;
        RETURN;
    1130:
        FuUnicodeCodepointCaseConvert := 1131;
        RETURN;
    1131:
        FuUnicodeCodepointCaseConvert := 1130;
        RETURN;
    1132:
        FuUnicodeCodepointCaseConvert := 1133;
        RETURN;
    1133:
        FuUnicodeCodepointCaseConvert := 1132;
        RETURN;
    1134:
        FuUnicodeCodepointCaseConvert := 1135;
        RETURN;
    1135:
        FuUnicodeCodepointCaseConvert := 1134;
        RETURN;
    1136:
        FuUnicodeCodepointCaseConvert := 1137;
        RETURN;
    1137:
        FuUnicodeCodepointCaseConvert := 1136;
        RETURN;
    1138:
        FuUnicodeCodepointCaseConvert := 1139;
        RETURN;
    1139:
        FuUnicodeCodepointCaseConvert := 1138;
        RETURN;
    1140:
        FuUnicodeCodepointCaseConvert := 1141;
        RETURN;
    1141:
        FuUnicodeCodepointCaseConvert := 1140;
        RETURN;
    1142:
        FuUnicodeCodepointCaseConvert := 1143;
        RETURN;
    1143:
        FuUnicodeCodepointCaseConvert := 1142;
        RETURN;
    1144:
        FuUnicodeCodepointCaseConvert := 1145;
        RETURN;
    1145:
        FuUnicodeCodepointCaseConvert := 1144;
        RETURN;
    1146:
        FuUnicodeCodepointCaseConvert := 1147;
        RETURN;
    1147:
        FuUnicodeCodepointCaseConvert := 1146;
        RETURN;
    1148:
        FuUnicodeCodepointCaseConvert := 1149;
        RETURN;
    1149:
        FuUnicodeCodepointCaseConvert := 1148;
        RETURN;
    1150:
        FuUnicodeCodepointCaseConvert := 1151;
        RETURN;
    1151:
        FuUnicodeCodepointCaseConvert := 1150;
        RETURN;
    1152:
        FuUnicodeCodepointCaseConvert := 1153;
        RETURN;
    1153:
        FuUnicodeCodepointCaseConvert := 1152;
        RETURN;
    1162:
        FuUnicodeCodepointCaseConvert := 1163;
        RETURN;
    1163:
        FuUnicodeCodepointCaseConvert := 1162;
        RETURN;
    1164:
        FuUnicodeCodepointCaseConvert := 1165;
        RETURN;
    1165:
        FuUnicodeCodepointCaseConvert := 1164;
        RETURN;
    1166:
        FuUnicodeCodepointCaseConvert := 1167;
        RETURN;
    1167:
        FuUnicodeCodepointCaseConvert := 1166;
        RETURN;
    1168:
        FuUnicodeCodepointCaseConvert := 1169;
        RETURN;
    1169:
        FuUnicodeCodepointCaseConvert := 1168;
        RETURN;
    1170:
        FuUnicodeCodepointCaseConvert := 1171;
        RETURN;
    1171:
        FuUnicodeCodepointCaseConvert := 1170;
        RETURN;
    1172:
        FuUnicodeCodepointCaseConvert := 1173;
        RETURN;
    1173:
        FuUnicodeCodepointCaseConvert := 1172;
        RETURN;
    1174:
        FuUnicodeCodepointCaseConvert := 1175;
        RETURN;
    1175:
        FuUnicodeCodepointCaseConvert := 1174;
        RETURN;
    1176:
        FuUnicodeCodepointCaseConvert := 1177;
        RETURN;
    1177:
        FuUnicodeCodepointCaseConvert := 1176;
        RETURN;
    1178:
        FuUnicodeCodepointCaseConvert := 1179;
        RETURN;
    1179:
        FuUnicodeCodepointCaseConvert := 1178;
        RETURN;
    1180:
        FuUnicodeCodepointCaseConvert := 1181;
        RETURN;
    1181:
        FuUnicodeCodepointCaseConvert := 1180;
        RETURN;
    1182:
        FuUnicodeCodepointCaseConvert := 1183;
        RETURN;
    1183:
        FuUnicodeCodepointCaseConvert := 1182;
        RETURN;
    1184:
        FuUnicodeCodepointCaseConvert := 1185;
        RETURN;
    1185:
        FuUnicodeCodepointCaseConvert := 1184;
        RETURN;
    1186:
        FuUnicodeCodepointCaseConvert := 1187;
        RETURN;
    1187:
        FuUnicodeCodepointCaseConvert := 1186;
        RETURN;
    1188:
        FuUnicodeCodepointCaseConvert := 1189;
        RETURN;
    1189:
        FuUnicodeCodepointCaseConvert := 1188;
        RETURN;
    1190:
        FuUnicodeCodepointCaseConvert := 1191;
        RETURN;
    1191:
        FuUnicodeCodepointCaseConvert := 1190;
        RETURN;
    1192:
        FuUnicodeCodepointCaseConvert := 1193;
        RETURN;
    1193:
        FuUnicodeCodepointCaseConvert := 1192;
        RETURN;
    1194:
        FuUnicodeCodepointCaseConvert := 1195;
        RETURN;
    1195:
        FuUnicodeCodepointCaseConvert := 1194;
        RETURN;
    1196:
        FuUnicodeCodepointCaseConvert := 1197;
        RETURN;
    1197:
        FuUnicodeCodepointCaseConvert := 1196;
        RETURN;
    1198:
        FuUnicodeCodepointCaseConvert := 1199;
        RETURN;
    1199:
        FuUnicodeCodepointCaseConvert := 1198;
        RETURN;
    1200:
        FuUnicodeCodepointCaseConvert := 1201;
        RETURN;
    1201:
        FuUnicodeCodepointCaseConvert := 1200;
        RETURN;
    1202:
        FuUnicodeCodepointCaseConvert := 1203;
        RETURN;
    1203:
        FuUnicodeCodepointCaseConvert := 1202;
        RETURN;
    1204:
        FuUnicodeCodepointCaseConvert := 1205;
        RETURN;
    1205:
        FuUnicodeCodepointCaseConvert := 1204;
        RETURN;
    1206:
        FuUnicodeCodepointCaseConvert := 1207;
        RETURN;
    1207:
        FuUnicodeCodepointCaseConvert := 1206;
        RETURN;
    1208:
        FuUnicodeCodepointCaseConvert := 1209;
        RETURN;
    1209:
        FuUnicodeCodepointCaseConvert := 1208;
        RETURN;
    1210:
        FuUnicodeCodepointCaseConvert := 1211;
        RETURN;
    1211:
        FuUnicodeCodepointCaseConvert := 1210;
        RETURN;
    1212:
        FuUnicodeCodepointCaseConvert := 1213;
        RETURN;
    1213:
        FuUnicodeCodepointCaseConvert := 1212;
        RETURN;
    1214:
        FuUnicodeCodepointCaseConvert := 1215;
        RETURN;
    1215:
        FuUnicodeCodepointCaseConvert := 1214;
        RETURN;
    1216:
        FuUnicodeCodepointCaseConvert := 1231;
        RETURN;
    1217:
        FuUnicodeCodepointCaseConvert := 1218;
        RETURN;
    1218:
        FuUnicodeCodepointCaseConvert := 1217;
        RETURN;
    1219:
        FuUnicodeCodepointCaseConvert := 1220;
        RETURN;
    1220:
        FuUnicodeCodepointCaseConvert := 1219;
        RETURN;
    1221:
        FuUnicodeCodepointCaseConvert := 1222;
        RETURN;
    1222:
        FuUnicodeCodepointCaseConvert := 1221;
        RETURN;
    1223:
        FuUnicodeCodepointCaseConvert := 1224;
        RETURN;
    1224:
        FuUnicodeCodepointCaseConvert := 1223;
        RETURN;
    1225:
        FuUnicodeCodepointCaseConvert := 1226;
        RETURN;
    1226:
        FuUnicodeCodepointCaseConvert := 1225;
        RETURN;
    1227:
        FuUnicodeCodepointCaseConvert := 1228;
        RETURN;
    1228:
        FuUnicodeCodepointCaseConvert := 1227;
        RETURN;
    1229:
        FuUnicodeCodepointCaseConvert := 1230;
        RETURN;
    1230:
        FuUnicodeCodepointCaseConvert := 1229;
        RETURN;
    1231:
        FuUnicodeCodepointCaseConvert := 1216;
        RETURN;
    1232:
        FuUnicodeCodepointCaseConvert := 1233;
        RETURN;
    1233:
        FuUnicodeCodepointCaseConvert := 1232;
        RETURN;
    1234:
        FuUnicodeCodepointCaseConvert := 1235;
        RETURN;
    1235:
        FuUnicodeCodepointCaseConvert := 1234;
        RETURN;
    1236:
        FuUnicodeCodepointCaseConvert := 1237;
        RETURN;
    1237:
        FuUnicodeCodepointCaseConvert := 1236;
        RETURN;
    1238:
        FuUnicodeCodepointCaseConvert := 1239;
        RETURN;
    1239:
        FuUnicodeCodepointCaseConvert := 1238;
        RETURN;
    1240:
        FuUnicodeCodepointCaseConvert := 1241;
        RETURN;
    1241:
        FuUnicodeCodepointCaseConvert := 1240;
        RETURN;
    1242:
        FuUnicodeCodepointCaseConvert := 1243;
        RETURN;
    1243:
        FuUnicodeCodepointCaseConvert := 1242;
        RETURN;
    1244:
        FuUnicodeCodepointCaseConvert := 1245;
        RETURN;
    1245:
        FuUnicodeCodepointCaseConvert := 1244;
        RETURN;
    1246:
        FuUnicodeCodepointCaseConvert := 1247;
        RETURN;
    1247:
        FuUnicodeCodepointCaseConvert := 1246;
        RETURN;
    1248:
        FuUnicodeCodepointCaseConvert := 1249;
        RETURN;
    1249:
        FuUnicodeCodepointCaseConvert := 1248;
        RETURN;
    1250:
        FuUnicodeCodepointCaseConvert := 1251;
        RETURN;
    1251:
        FuUnicodeCodepointCaseConvert := 1250;
        RETURN;
    1252:
        FuUnicodeCodepointCaseConvert := 1253;
        RETURN;
    1253:
        FuUnicodeCodepointCaseConvert := 1252;
        RETURN;
    1254:
        FuUnicodeCodepointCaseConvert := 1255;
        RETURN;
    1255:
        FuUnicodeCodepointCaseConvert := 1254;
        RETURN;
    1256:
        FuUnicodeCodepointCaseConvert := 1257;
        RETURN;
    1257:
        FuUnicodeCodepointCaseConvert := 1256;
        RETURN;
    1258:
        FuUnicodeCodepointCaseConvert := 1259;
        RETURN;
    1259:
        FuUnicodeCodepointCaseConvert := 1258;
        RETURN;
    1260:
        FuUnicodeCodepointCaseConvert := 1261;
        RETURN;
    1261:
        FuUnicodeCodepointCaseConvert := 1260;
        RETURN;
    1262:
        FuUnicodeCodepointCaseConvert := 1263;
        RETURN;
    1263:
        FuUnicodeCodepointCaseConvert := 1262;
        RETURN;
    1264:
        FuUnicodeCodepointCaseConvert := 1265;
        RETURN;
    1265:
        FuUnicodeCodepointCaseConvert := 1264;
        RETURN;
    1266:
        FuUnicodeCodepointCaseConvert := 1267;
        RETURN;
    1267:
        FuUnicodeCodepointCaseConvert := 1266;
        RETURN;
    1268:
        FuUnicodeCodepointCaseConvert := 1269;
        RETURN;
    1269:
        FuUnicodeCodepointCaseConvert := 1268;
        RETURN;
    1270:
        FuUnicodeCodepointCaseConvert := 1271;
        RETURN;
    1271:
        FuUnicodeCodepointCaseConvert := 1270;
        RETURN;
    1272:
        FuUnicodeCodepointCaseConvert := 1273;
        RETURN;
    1273:
        FuUnicodeCodepointCaseConvert := 1272;
        RETURN;
    1274:
        FuUnicodeCodepointCaseConvert := 1275;
        RETURN;
    1275:
        FuUnicodeCodepointCaseConvert := 1274;
        RETURN;
    1276:
        FuUnicodeCodepointCaseConvert := 1277;
        RETURN;
    1277:
        FuUnicodeCodepointCaseConvert := 1276;
        RETURN;
    1278:
        FuUnicodeCodepointCaseConvert := 1279;
        RETURN;
    1279:
        FuUnicodeCodepointCaseConvert := 1278;
        RETURN;
    1280:
        FuUnicodeCodepointCaseConvert := 1281;
        RETURN;
    1281:
        FuUnicodeCodepointCaseConvert := 1280;
        RETURN;
    1282:
        FuUnicodeCodepointCaseConvert := 1283;
        RETURN;
    1283:
        FuUnicodeCodepointCaseConvert := 1282;
        RETURN;
    1284:
        FuUnicodeCodepointCaseConvert := 1285;
        RETURN;
    1285:
        FuUnicodeCodepointCaseConvert := 1284;
        RETURN;
    1286:
        FuUnicodeCodepointCaseConvert := 1287;
        RETURN;
    1287:
        FuUnicodeCodepointCaseConvert := 1286;
        RETURN;
    1288:
        FuUnicodeCodepointCaseConvert := 1289;
        RETURN;
    1289:
        FuUnicodeCodepointCaseConvert := 1288;
        RETURN;
    1290:
        FuUnicodeCodepointCaseConvert := 1291;
        RETURN;
    1291:
        FuUnicodeCodepointCaseConvert := 1290;
        RETURN;
    1292:
        FuUnicodeCodepointCaseConvert := 1293;
        RETURN;
    1293:
        FuUnicodeCodepointCaseConvert := 1292;
        RETURN;
    1294:
        FuUnicodeCodepointCaseConvert := 1295;
        RETURN;
    1295:
        FuUnicodeCodepointCaseConvert := 1294;
        RETURN;
    1296:
        FuUnicodeCodepointCaseConvert := 1297;
        RETURN;
    1297:
        FuUnicodeCodepointCaseConvert := 1296;
        RETURN;
    1298:
        FuUnicodeCodepointCaseConvert := 1299;
        RETURN;
    1299:
        FuUnicodeCodepointCaseConvert := 1298;
        RETURN;
    1300:
        FuUnicodeCodepointCaseConvert := 1301;
        RETURN;
    1301:
        FuUnicodeCodepointCaseConvert := 1300;
        RETURN;
    1302:
        FuUnicodeCodepointCaseConvert := 1303;
        RETURN;
    1303:
        FuUnicodeCodepointCaseConvert := 1302;
        RETURN;
    1304:
        FuUnicodeCodepointCaseConvert := 1305;
        RETURN;
    1305:
        FuUnicodeCodepointCaseConvert := 1304;
        RETURN;
    1306:
        FuUnicodeCodepointCaseConvert := 1307;
        RETURN;
    1307:
        FuUnicodeCodepointCaseConvert := 1306;
        RETURN;
    1308:
        FuUnicodeCodepointCaseConvert := 1309;
        RETURN;
    1309:
        FuUnicodeCodepointCaseConvert := 1308;
        RETURN;
    1310:
        FuUnicodeCodepointCaseConvert := 1311;
        RETURN;
    1311:
        FuUnicodeCodepointCaseConvert := 1310;
        RETURN;
    1312:
        FuUnicodeCodepointCaseConvert := 1313;
        RETURN;
    1313:
        FuUnicodeCodepointCaseConvert := 1312;
        RETURN;
    1314:
        FuUnicodeCodepointCaseConvert := 1315;
        RETURN;
    1315:
        FuUnicodeCodepointCaseConvert := 1314;
        RETURN;
    1316:
        FuUnicodeCodepointCaseConvert := 1317;
        RETURN;
    1317:
        FuUnicodeCodepointCaseConvert := 1316;
        RETURN;
    1318:
        FuUnicodeCodepointCaseConvert := 1319;
        RETURN;
    1319:
        FuUnicodeCodepointCaseConvert := 1318;
        RETURN;
    1320:
        FuUnicodeCodepointCaseConvert := 1321;
        RETURN;
    1321:
        FuUnicodeCodepointCaseConvert := 1320;
        RETURN;
    1322:
        FuUnicodeCodepointCaseConvert := 1323;
        RETURN;
    1323:
        FuUnicodeCodepointCaseConvert := 1322;
        RETURN;
    1324:
        FuUnicodeCodepointCaseConvert := 1325;
        RETURN;
    1325:
        FuUnicodeCodepointCaseConvert := 1324;
        RETURN;
    1326:
        FuUnicodeCodepointCaseConvert := 1327;
        RETURN;
    1327:
        FuUnicodeCodepointCaseConvert := 1326;
        RETURN;
    1329:
        FuUnicodeCodepointCaseConvert := 1377;
        RETURN;
    1330:
        FuUnicodeCodepointCaseConvert := 1378;
        RETURN;
    1331:
        FuUnicodeCodepointCaseConvert := 1379;
        RETURN;
    1332:
        FuUnicodeCodepointCaseConvert := 1380;
        RETURN;
    1333:
        FuUnicodeCodepointCaseConvert := 1381;
        RETURN;
    1334:
        FuUnicodeCodepointCaseConvert := 1382;
        RETURN;
    1335:
        FuUnicodeCodepointCaseConvert := 1383;
        RETURN;
    1336:
        FuUnicodeCodepointCaseConvert := 1384;
        RETURN;
    1337:
        FuUnicodeCodepointCaseConvert := 1385;
        RETURN;
    1338:
        FuUnicodeCodepointCaseConvert := 1386;
        RETURN;
    1339:
        FuUnicodeCodepointCaseConvert := 1387;
        RETURN;
    1340:
        FuUnicodeCodepointCaseConvert := 1388;
        RETURN;
    1341:
        FuUnicodeCodepointCaseConvert := 1389;
        RETURN;
    1342:
        FuUnicodeCodepointCaseConvert := 1390;
        RETURN;
    1343:
        FuUnicodeCodepointCaseConvert := 1391;
        RETURN;
    1344:
        FuUnicodeCodepointCaseConvert := 1392;
        RETURN;
    1345:
        FuUnicodeCodepointCaseConvert := 1393;
        RETURN;
    1346:
        FuUnicodeCodepointCaseConvert := 1394;
        RETURN;
    1347:
        FuUnicodeCodepointCaseConvert := 1395;
        RETURN;
    1348:
        FuUnicodeCodepointCaseConvert := 1396;
        RETURN;
    1349:
        FuUnicodeCodepointCaseConvert := 1397;
        RETURN;
    1350:
        FuUnicodeCodepointCaseConvert := 1398;
        RETURN;
    1351:
        FuUnicodeCodepointCaseConvert := 1399;
        RETURN;
    1352:
        FuUnicodeCodepointCaseConvert := 1400;
        RETURN;
    1353:
        FuUnicodeCodepointCaseConvert := 1401;
        RETURN;
    1354:
        FuUnicodeCodepointCaseConvert := 1402;
        RETURN;
    1355:
        FuUnicodeCodepointCaseConvert := 1403;
        RETURN;
    1356:
        FuUnicodeCodepointCaseConvert := 1404;
        RETURN;
    1357:
        FuUnicodeCodepointCaseConvert := 1405;
        RETURN;
    1358:
        FuUnicodeCodepointCaseConvert := 1406;
        RETURN;
    1359:
        FuUnicodeCodepointCaseConvert := 1407;
        RETURN;
    1360:
        FuUnicodeCodepointCaseConvert := 1408;
        RETURN;
    1361:
        FuUnicodeCodepointCaseConvert := 1409;
        RETURN;
    1362:
        FuUnicodeCodepointCaseConvert := 1410;
        RETURN;
    1363:
        FuUnicodeCodepointCaseConvert := 1411;
        RETURN;
    1364:
        FuUnicodeCodepointCaseConvert := 1412;
        RETURN;
    1365:
        FuUnicodeCodepointCaseConvert := 1413;
        RETURN;
    1366:
        FuUnicodeCodepointCaseConvert := 1414;
        RETURN;
    1377:
        FuUnicodeCodepointCaseConvert := 1329;
        RETURN;
    1378:
